# B&R Automation Studio project TD52 (part 110)

#### biogasCyclic.st - Cyclic code
```iecst
(*
***************************************************************************
biogas			control/monitoring gas blower/flare

This code is confidential and proprietary to the INNIO Company.
It may not be used in any form, or reproduced in any manner,
without the express written permission of the INNIO Company.
Copyright, INNIO Company, 2025

Customized modifications: -
------------------------

History:
-------
V0.0		03.12.05/LH	erstellt
V2071		02.02.05/LH	angepasst für V2.071
 			03.03.05/LH	angepasst für neue Gasdrucküberwachungsphilosophie
V2072		16.11.05/LH	angepasst für Modulisierung
V2201		08.08.07/LH	Vorhalte Gasverdichter vor Öffnen 1. Gasstr. während Gasumschaltung
 			12.09.07/LH	Freigabe Fackel nur wenn Gasverdichter nicht gestört ist
V2600		06.08.2009 lettenb.	task activation added
V3.10.0		15.02.2010 lettenb.	QUITT_AB, IN_GT.tAB2GT replaced by reset_alarm[x], quitt_wa
V3.20.0		17.01.2011 lettenb.	connections to alarmsXXxx added, user comment
			14.02.2011	release main gas valve FG_HGV moved to task pb8, enable alarms added
V3.99		21.09.2013	Ganguly/Denk, generated for modular software
V3.99.1		19.09.2013	Denk, V3.30.0 and V3.30.2 changes inserted
V3.99.2		25.03.2013	pankajrodey, Integration for 3.40
V4.03.00	15.03.2016	Denk, Bugfix Alarm Set for A3317
			04.04.2016	Denk, Bugfix Alarm Set for A3328
V4.04.00	26-10-2016	Denk, Logic change for gastemperature messages 3317 and 3568
V4.07.00	19.03.2019	Zengerer, Demand compressor options for TKE Gastrain Types
V4.07.01	16.10.2019	Zengerer, Demand compressor option TOF bMEGA_GasTrain, Operating message: B2997 extended compressor demand for gas leakage check
V4.07.02	25.10.2019	Zengerer  EDGEPOS(OUT_GT.tGT1_SafeDevice.Do) takeover from V4.07 Basisupdate
V4.09.00	16.01.2020	Zengerer  bDelayGDKG_GCStarting to delay leakage check, to allow gas compressor generate sufficient pressure, bDem_SafeDevice	(corr.Jan2020)
			06.02.2020	Zengerer  bMsg2997_Set changed, avaid  GC restart after failure reset
V4.25.00	17.12.2025	Tinello   Safety signals added

Instructions for use:
--------------------
 - activate task if used (see comment)
 - disable gas blower if not existing
 - RM "Fackel in Betrieb" in fb31_hb einbinden und in BILD_50 zur Anzeige bringen!

enable biogas alarms in the specific network if used:			default:

A3316	Gas compressor failure					active
W3567	Gas compressor failure					not active

A3317	Gas temperature high					active
W3568	Gas temperature high					not active
A3328 	Gas temperature measuring signal failure				not active

A3318	Gas pressure low before compressor				active
W3569	Gas pressure low before gas compressor				not active
A3327	Gas pressure before gas compressor measuring signal failure		not active
W3570	Gas pressure before gas compressor measuring signal failure		not active

A3326	Idle operation time gas compressor maximum			active

W3520	Flare failure						active

Outstandings:
------------
*********************************************

*)

PROGRAM _CYCLIC

IF NOT Para.bBiogasActive THEN
	bDelayGDKG_GCStarting := FALSE;				(*inactive bigas compressor should not delay  bDelayGDKG_GCStarting leakage check*)
	RETURN;
ELSE

	(* Alarm Set for A3327: Measurement signal error Gas pressure before compressor *)
	bMsg3327_Set := Para.bMsg3327Active AND NOT IN_GT.tPr_GT_Suct.GoodQual AND NOT OUT_GT.bGT2_Select;

	(* Alarm Set for W3570: Measurement signal error Gas pressure before compressor *)
	bMsg3570_Set := Para.bMsg3570Active AND NOT IN_GT.tPr_GT_Suct.GoodQual AND NOT MM2VIS.bMsg3327 AND NOT bMsg3327_Set;

	(* Alarm Set for A3318 Gas pressure minimum before compressor *)
	xTON_FA_ZM_GDMI11.IN := MM2VIS.bMsgDummy_Min_SuctPr OR NOT IN_GT.tPr_GT_MinBefCompr.Di;
	xTON_FA_ZM_GDMI11.PT := T#2s;
	xTON_FA_ZM_GDMI11();
	HM_GDMI11    := xTON_FA_ZM_GDMI11.Q;
	bMsg3318_Set := HM_GDMI11 AND ((FG_GDRUW AND NOT OUT_GT.bGT2_Select) OR bMsg3318_Set);

	(* Alarm Set for W3569 Gas pressure minimum before compressor maximum *)
	bMsg3569_Set := Para.bMsg3569Active
		            AND HM_GDMI11
		            AND NOT MM2VIS.bMsg3318
		            AND NOT bMsg3318_Set
		            AND Para.bGCActive
		            AND (OUT_GT.bGT_TypSwhActive OR OUT_GT.bGT_TypSwhActiveHalt);

	(* Alarm Set for A3328: Measurement signal from "spec_gas"*)
	bMsg3328_Set := Para.bMsg3328Active AND NOT IN_GT.tT_GT.GoodQual AND NOT OUT_GT.bGT2_Select;

	(* Alarm Set for A3317 Gas temperature maximum *)
	bMsg3317_Set := ((GT_MAX AND IN_GT.tT_GT.GoodQual) OR NOT IN_GT.tT_GT_Ok.Di) AND NOT OUT_GT.bGT2_Select;

	(* Alarm Set for W3568: Gas temperature maximum *)
	bMsg3568_Set := Para.bMsg3568Active AND ((GT_MAX AND IN_GT.tT_GT.GoodQual) OR NOT IN_GT.tT_GT_Ok.Di) AND NOT MM2VIS.bMsg3317 AND NOT bMsg3317_Set;

	(* Alarm Set  for A3316: Trip: Gas compressor failure *)
	bMsg3316_Set := NOT IN_GT.tGT_GC_Fail.Di AND NOT OUT_GT.bGT2_Select;

	(* Alarm Set for W3567: Warning: Gas compressor failure *)
	bMsg3567_Set := Para.bMsg3567Active AND NOT IN_GT.tGT_GC_Fail.Di AND NOT MM2VIS.bMsg3316 AND NOT bMsg3316_Set;

	(* Flare failure *)
	bMsg3520_Set := NOT IN_GT.tGT_FlairFail.Di;

	IF (bMEGA_GasTrain) THEN					(*derived from option bit2 = '4' == MEGA Gas Train, for wide pipe dimensions with 2 separate valves 	(V4.07	Requisition- supplied code parts included for MGV) *)
		(* Demand compressor for Module operation *)
		(*-------------------------------------------------------------------------------------*)
		TOF_MEGA_GC.IN := EDGEPOS(NOT IN_GT.bSafetyPLC_Active AND bDem_SafeDevice)  						// V4.07 Basisupdate 2  old: EDGEPOS(OUT_GT.tGT1_SafeDevice.Do);(* SAFETY PLC *)
						  OR	 (	  IN_GT.bSafetyPLC_Active AND IN_GT.tSafetyLoop_Eng.Di AND NOT IN_GT.bSafeOUT_GT1_SD_Dem_PS); 											(* SAFETY PLC *)

		IF IN_GT.tAB2GT.bGnlTrip1 OR  IN_GT.tAB2GT.bGnlTrip2 OR OUT_GT.bMsg1027 THEN 						// OR IN_GT.tAB2GT.bGnlTrip3 THEN
			TOF_MEGA_GC.PT := 0 ;									// V4.09: avoid  GC restart after failure reset
		ELSE
			TOF_MEGA_GC.PT := IN_GT.tCU2GT.tiGT_TestDuration; 		// T#120s;	 (*time for gas compressor / Gas sfety check [s] *)
		END_IF

		TOF_MEGA_GC();
		(*-------------------------------------------------------------------------------------*)
		bDem_GC_M :=   (IN_GT.bEng_Aux_Dem OR (TOF_MEGA_GC.Q AND NOT IN_GT.tGT1_SafeDevOK.Di AND NOT IN_GT.bSafeOUT_GT1_SafeDevOK))	(*gas compressor demand extension*) 	(* SAFETY PLC *)
				AND NOT IN_GT.bMsg1053
				AND NOT IN_GT.bMsg1054
				AND NOT IN_GT.bMsg1031
				AND NOT OUT_GT.bGT2_Select;

		bMsg2997_Set := Para.bGCActive
				AND OUT_GT.tGT_GC_Dem.Do
				AND bDem_GC_M
				AND NOT IN_GT.tEng_Run.Do
				AND NOT IN_GT.bEng_Aux_Dem
				AND NOT IN_GT.tGT1_SafeDevOK.Di ;
				// := 	Para.bGCActive AND  OUT_GT.tGT_GC_Dem.Do  AND TOF_MEGA_GC.Q	; 		(* Megagas Operating message: B2997 gas compressor demand extension - gas leakage test (new in V4.09)*)

	ELSE
		(* Demand compressor for Module operation *)
		bDem_GC_M := IN_GT.bEng_Aux_Dem 							//OLD: gas compressor demand intermediate  ANF_V_M :=
				AND NOT IN_GT.bMsg1053
				AND NOT IN_GT.bMsg1054
				AND NOT IN_GT.bMsg1031
				AND NOT OUT_GT.bGT2_Select;
	END_IF

		(* Demand Flair *)
	ANF_FA :=	IN_GT.tDemFlair.Di AND NOT IN_GT.bMsg1053 AND NOT IN_GT.bMsg1054 AND NOT IN_GT.bMsg1031
	            AND NOT bDem_GC_M AND IN_GT.tFlairRdy.Di AND NOT MM2VIS.bMsg3520;

	(* Release  Flare (only when Gas compressure has not failed *)
	xTON_FG_FA.IN := IN_GT.tGT_GC_Fail.Di ;
	xTON_FG_FA.PT := T#5s;
	xTON_FG_FA();
	OUT_GT.tGT_RelFlair.Do := xTON_FG_FA.Q AND ANF_FA;

	(* Demand gas compressor *)
	ANF_GVD_1				:=	ANF_FA
	           					OR (bDem_GC_M AND (OUT_GT.tGV1_Open.Do OR V_GVD OR NOT IN_GT.tEng_Run.Do));
	OUT_GT.tGT_GC_Dem.Do 	:= FG_HGV AND ANF_GVD_1 AND NOT MM2VIS.bMsg3318 AND NOT MM2VIS.bMsg3221 AND NOT MM2VIS.bMsg3327 AND NOT MM2VIS.bMsg3326 AND NOT MM2VIS.bMsg3316;

	(* Monitoring idle operation time gas compressor maximum *)
	bMsg3326_Set := OUT_GT.tGT_GC_Dem.Do
					AND ((NOT IN_GT.tEng_Run.Do AND bDem_GC_M) OR (OUT_GT.tGT_RelFlair.Do AND NOT IN_GT.tGT_FlareOpMod.Di));

	(* Release gas pressure monitoring (Gas pressure minimum Gas train 1 (p10_1001)) *)
	xTON_FA_GASV1.IN := OUT_GT.tGV1_Open.Do;
	xTON_FA_GASV1.PT := Para.tiGT1_Delay_Mon;			// 5s parameter introduced in V3.30
	xTON_FA_GASV1();

	xTON_FA_T_GDRUW.IN := IN_GT.bEng_Aux_Dem OR ((bDem_SafeDevice OR NOT IN_GT.bSafeOUT_GT1_SafeDevOK) AND OUT_GT.tGT_GC_Dem.Do);	(*Engine Demand OR Gas Safety Check Demand*)	(* SAFETY PLC *)
	xTON_FA_T_GDRUW.PT := Para.tiGT1_Delay_Mon;			// 5s parameter introduced in V3.30
	xTON_FA_T_GDRUW();

	T_GDRUW := (xTON_FA_GASV1.Q AND IN_GT.tEng_Run.Do) OR (xTON_FA_T_GDRUW.Q AND NOT IN_GT.tEng_Run.Do);

	(*generate flag to delay gas leakage checking*)
	xTOFDelayGDKG_GCStarting.IN	:= EDGEPOS(OUT_GT.tGT_GC_Dem.Do AND NOT IN_GT.tGT1_SafeDevOK.Di);  	(*bit to delay leakage check, to allow time for gas compressor building up sufficient pressure*)

	xTOFDelayGDKG_GCStarting(PT:= T#6s);
	bDelayGDKG_GCStarting 	:=xTOFDelayGDKG_GCStarting.Q ;
END_IF;

END_PROGRAM
```

#### biogas.var - Local variables
```iecst
(********************************************************************
 * COPYRIGHT -- INNIO Company
 ********************************************************************
 * Program: biogas
 * File: biogas.var
 * Author: 105051626
 * Created: April 19, 2012
 ********************************************************************
 * Local variables of program biogas
 ********************************************************************)
VAR
	ANF_FA : BOOL := 0; (* Anforderung Fackel *)
	bDem_GC_M : BOOL; (*Intermediate variable for Demand gas compressor*) (*OldName: ANF_V_M*)
	HM_GDMI11 : BOOL; (*Gas pressure minimum before compresssor*)
	ANF_GVD_1 : BOOL; (*Intermediate variable for interlocks of Demand gas compressor*)
	xTON_FA_ZM_GDMI11 : TON;
	xTON_FA_GASV1 : TON;
	xTON_FG_FA : TON;
	xTON_FA_T_GDRUW : TON;
	TOF_MEGA_GC : TOF; (*Gas compressor timer for Mega Gasvalve option*)
	xTOFDelayGDKG_GCStarting : TOF; (*prevent saftey device reaction to low gas pressure*)
END_VAR
```

### Program Logical/Gastrain/bm3_nm3 (IEC) - bm3_mn3

#### bm3_nm3Cyclic.st - Cyclic code
```iecst
(* BERECHNUNG NORMKUBIKMETER-GASVERBRAUCH

VER	Datum/Name	Änderung
V170	21.03.02/LH	erstellt
V172	31.07.02/LH	Gaszähler-Impuls aus pb7 übernommen
					Berechnung Zustandszahl eliminiert => neuer task
		17.09.02/LH	korrigiert für AS 2.2
V173	11.11.02/LH	Vergleich korrigiert
V181	23.04.03/LH	Zähler-Beschaltung richtiggestellt
V190	18.06.04/LH	Vermeidung von Rundungsfehlern
V03.99.00	21.09.2013	Ganguly/Denk 	Generated for modular software
V04.00.02	02.06.2014  Denk			Gas counter to MM2VIS added
V04.01.00	01.07.2014  Denk			Gas counter parameters added and additional OUT-Interfaces
V04.01.01	18.03.2015	lettenb.		increase counter with NORM_IMP, xR_TRIG_FA_BTRB_IMP.Q only for 1 cycle
V04.03.00	02.06.2015	Denk			Bugfix, gas counter reset when PLC coldstart. Connected to Perm struct.
V04.04.00	18.10.2016	Denk			Gas counter writable from Visu
V04.07.00	10.04.2019	Zengerer		Gas counter prescaler for requisition demanded version V4.07, chapter 5
V04.07.01	11.04.2019	Zengerer		xTOF_FA_BTRB_M3.PT := ...tiGCPulse_Duration_min
V04.07.02	05.06.2019	Zengerer		cleanup, disabeled xCTD_FA_GAS_IMP removed

Instructions FOR use:
--------------------
 -

Outstandings:
------------
rGasImp_Prescaling < 1.0 ..  //TODO:Release after pilot engines in V4.09

**********************************************)

PROGRAM _CYCLIC

    (* Reset Nm3-Impulse *)
	NORM_IMP := FALSE;

	(* Gas counter - impulse *)

	IF IN_GT.tCU2GT.iGC_Select_Option.7  THEN 					// Bit 7 sets task input back to behavior of former task version <4.07
		xR_TRIG_FA_GAS_IMP_CD.CLK := IN_GT.tCnt_GasImp.Di;		// Direct DI input like in former task version <4.07
	ELSE
		xR_TRIG_FA_GAS_IMP_CD.CLK := bGasImp_Prescaled;			// Pulse prescaler for IN_GT.tCnt_GasImp.Di gets handled in TC2
	END_IF
	xR_TRIG_FA_GAS_IMP_CD();
	IF NOT IN_GT.tCnt_GasImp.Di THEN bGasImp_Prescaled := FALSE; END_IF	(* Do not clear the artificial generated pulse, until the real pulse is gone, to keep similar pulse duration behavior *)

	BTRB_IMP   := xR_TRIG_FA_GAS_IMP_CD.Q AND ANLAUF;

	ANLAUF := TRUE;											// Setting local flag to TRUE , it is initially FALSE

	(* Bm3-Impulse *)
	xTOF_FA_BTRB_M3.IN := BTRB_IMP;
	xTOF_FA_BTRB_M3.PT := IN_GT.tCU2GT.tiGCPulse_Duration_min ;   		// := T#1s;
	xTOF_FA_BTRB_M3();
	BTRB_M3 := xTOF_FA_BTRB_M3.Q;

	(* Edge triggered Gas count impulse *)
	xR_TRIG_FA_BTRB_IMP.CLK := BTRB_M3;
	xR_TRIG_FA_BTRB_IMP();

	IMP_W := LIMIT(1000, Para.rGasImp_Prescaling * 1000, 50000);		 (*NEW parameter from V4.07: (Impulswertigkeit (Caution: formerly Constant value 1000 removed, but 1000 has to be FIXED LOWER LIMIT to cooperate with prescaler!)  *)

	IF xR_TRIG_FA_BTRB_IMP.Q THEN
		IMP_B := IMP_W;
	ELSE
		IMP_B := 0;
	END_IF;

	(* L10-L12 Summe *)
	IMP_N := ZSZ * IMP_B;

	(* Sum up impulses *)
	IMP_S := LIMIT(0, (IMP_S + IMP_N) ,4294967295);

	(* Block new impulse *)
	xTOF_FA_T_NORM_M3.IN := NORM_M3;
	xTOF_FA_T_NORM_M3.PT := IN_GT.tCU2GT.tiGCPulse_Duration_min ;   		// := T#1s;
	xTOF_FA_T_NORM_M3();
	T_NORM_M3 := xTOF_FA_T_NORM_M3.Q;

	(* Sum greater than impulse "wertigkeit" & release new impulse *)
	IF ((IMP_S >= IMP_W) AND NOT T_NORM_M3) THEN
		(* Set Nm3 impulse *)
		NORM_IMP := TRUE;
		(* Reduce sum by impulse "wertigkeit *)
		IMP_S := IMP_S - IMP_W;
	END_IF;

	(* Nm3 impulse *)
	xTOF_FA_NORM_M3.IN := NORM_IMP;
	xTOF_FA_NORM_M3.PT := IN_GT.tCU2GT.tiGCPulse_Duration_min ;   		// := T#1s;
	xTOF_FA_NORM_M3();
	NORM_M3 := xTOF_FA_NORM_M3.Q;

	(* Counter *)
	IF Para.bCnt_Gas_NormM3 THEN
		(* Gas counter Norm_M3 *)
		IF NORM_IMP THEN
			(* increase counter *)
			MM2VIS.iCnt_Gas_NormM3 := MM2VIS.iCnt_Gas_NormM3 + REAL_TO_DINT(MAX(1, Para.rGasImp_Prescaling));  // + 1; 	 Changed V4.07
			(* check limits *)
		ELSIF MM2VIS.iCnt_Gas_NormM3 >= 1000000000 THEN
			MM2VIS.iCnt_Gas_NormM3 := MM2VIS.iCnt_Gas_NormM3 - 1000000000;    (* check upper limit *)
		ELSIF MM2VIS.iCnt_Gas_NormM3 <= -1000000000 THEN
			MM2VIS.iCnt_Gas_NormM3 := MM2VIS.iCnt_Gas_NormM3 + 1000000000;    (* check lower limit *)
		END_IF;
	END_IF;

	IF Para.bCnt_Gas_OpM3 THEN
		(* Gas counter Op_M3 *)
		IF xR_TRIG_FA_BTRB_IMP.Q THEN
			(* increase counter *)
			MM2VIS.iCnt_Gas_OpM3 := MM2VIS.iCnt_Gas_OpM3 + REAL_TO_DINT(MAX(1, Para.rGasImp_Prescaling));  // + 1; 	 Changed V4.07
			(* check limits *)
		ELSIF MM2VIS.iCnt_Gas_OpM3 >= 1000000000 THEN
			MM2VIS.iCnt_Gas_OpM3 := MM2VIS.iCnt_Gas_OpM3 - 1000000000;        (* check upper limit *)
		ELSIF MM2VIS.iCnt_Gas_OpM3 <= -1000000000 THEN
			MM2VIS.iCnt_Gas_OpM3 := MM2VIS.iCnt_Gas_OpM3  + 1000000000;       (* check lower limit *)
		END_IF;
	END_IF;

	(* Assignement to OUT/MM2VIS-Interfaces *)
	OUT_GT.iCnt_Gas_OpM3   	:= MM2VIS.iCnt_Gas_OpM3;
	OUT_GT.iCnt_Gas_NormM3 	:= MM2VIS.iCnt_Gas_NormM3;
	OUT_GT.bCnt_Gas_OpM3   	:= BTRB_M3;
	OUT_GT.bCnt_Gas_NormM3 	:= NORM_M3;

END_PROGRAM
```

#### bm3_nm3.var - Local variables
```iecst
VAR
	ANLAUF : BOOL := 0;
	BTRB_IMP : BOOL := 0;
	BTRB_M3 : BOOL; (*Bm3 impulse   	CV_GAS_IMP : UINT := 0;	*)
	IMP_B : REAL;
	IMP_N : REAL;
	IMP_S : REAL; (* Impulssumme *)
	IMP_W : REAL; (* 1000 Impulswertigkeit (Caution: parameter value from V4.07 onward)*)
	NORM_IMP : BOOL;
	NORM_M3 : BOOL;
	T_NORM_M3 : BOOL := 0;  (*	xCTD_FA_GAS_IMP : CTD;  *)
	xR_TRIG_FA_BTRB_IMP : R_TRIG;
	xR_TRIG_FA_GAS_IMP_CD : R_TRIG;  (*	xR_TRIG_FA_GAS_IMP_LD : R_TRIG; *)
	xTOF_FA_BTRB_M3 : TOF;
	xTOF_FA_NORM_M3 : TOF;
	xTOF_FA_T_NORM_M3 : TOF;
END_VAR
```

### Program Logical/Gastrain/spec_gas (IEC) - spec_gas

#### spec_gasCyclic.st - Cyclic code
```iecst
(* MONITORING AND CONTROLING OF SPECIAL GAS ENGINES

variables (limit switches) for customized use:
 	GD_MAX	gas pressure maximum
 	GT_MAX	gas temperature maximum
 	GT_MIN	gas temperature minimum
 	SD_MAX	suction pressure maximum
 	SD_MIN	suction pressure minimum

MS_CV calorific value measuring signal failure
CV_MIN_A calorific value low
CV_MIN_W calorific value low
CV_RED reduction by calorific value active
OUT_GT.rP_Red_CV_Norm reduction value by calorific value

output variables to standard software:

BOOL:	CH4_MIN_A	--> A1086
 	CH4_MIN_W	--> W3154
 	FGGAS		--> W3153
 	GD_MIN_W	--> W3221
 	MS_CH4		--> W3155
 	MS_GD		--> W3156
 	MS_GM		--> W3160
 	MS_GT		--> W3159
 	MS_O2_A 	--> A1088
 	MS_O2_W 	--> W3158
 	MS_SD		--> W3157
 	O2_MAX		--> A1087

............................
VER	Datum/Name	Änderung
V180	19.11.02/LH	erstellt
V181	10.04.03/Th.	Korrekturen bei Typprüfung: OUT_GT.bGasSupplyOk
 	    11.04.03/Th.	Korrekturen bei Typprüfung: MS_O2_W, MS_O2_A
 	    17.04.03/Th.	Korrekturen bei Typprüfung: SD_MIN, SD_MAX
V183	16.10.03/LH	Messignal CH4-Gehalt erst aktiv mit IN_GT.bParaSetupOk
V184	07.01.04/ThJ	Messignalstörungen erst aktiv mit IN_GT.bParaSetupOk;
 			Reset CH4_MIN, MS_GM, MS_O2_A, MS_O2_W wenn nicht aktiviert.
 			Kommentare.
 			Zeitverz. für CH4_MIN 2 --> 5s.
V2071	30.11.04/LH	Korrektur Gasqualitätsberechnung
 	    03.02.05/LH	Überwachung Gasdruck minimum angepasst für V2071
 	    03.03.05/LH	Anpassung Saugdruck min/max
V2072	16.11.05/LH	CH4 min. / Gasdr. min. / Freigabe aus Gasstation lt. letzten Erkenntnissen angepasst
 			     Anforderung Entlastung eliminiert (wird nicht benötigt)
V190	19.03.04/LH	Interpolation GAS1_2 über Rezept einstellbar
 		    	 Leistungsreduktionen --> p_soll(classic)/powersel(XT)
 			     Umrechnungen --> ana_umr(classic)/ana_calc(XT)
V220	19.02.07/LH	angepasst für X20-Einführung
 	    01.03.07/LH	Erweiterung auf Pt100
 	    10.04.07/LH	Zuweisung für Pt100
V2.32	14.07.08/ThJ Heizwert/calorific value added
V2.34.0 04.12.2008 Lett./ThJ set GAS1_2 in case of Para.bGT_CVIpol12Active=true
V2.50.0	02.02.2009 lett. HW_WE -> AI_CV(for standard)
V03.99.00.00	21.09.2013	Ganguly	generated for modular software
V03.99.01.00	21.02.2013	Denk	Integration of V3.30 in modular software
									HM_GDMI1, HM_GDMI2 changed to modul global variable
V04.00.02.00	15.05.2014	Denk	Bugfix, FGGAS
V04.00.02.00	17.05.2014	Denk	Bugfix, Interpolations-Umschaltung, 4x Skalierung falsch 100% --> 1.0%
V04.01.00.00	17.07.2014	Denk	Bugfix, Measurement signal failure reset CH4 and CV signal
									Bugfix, Deactivation power reduction (CH4,GD,SD) via standard DI's
									Bugfix, CH4,CV: Para.rGT_CH4Mix1,Para.rGT_CH4Mix2 and Para.bGT_CVIpol12Active
V04.01.01.00	24.08.2014	Denk	Bugfix, Interpolation deactivation
V04.01.02.00	14.10.2014	Denk	Bugfix, Message activation O2 max.
V04.03.00.00	31.03.2015	Denk	Improvement, additional LABELS for tPr_GT1_1_Min and tPr_GT1_1_Max
				02.07.2015	Denk 	Bugfix, 3221 not activ when gastrain 2 is active. NOT was missing. NOT MM2VIS.bMsg1028
									Warnings for 4 gaslines bMsg2694-2696 added
V04.10.0.00		08.12.2020	Denk	Bugfix, xTON_GDMA2() changed to xTON_GDMA2_VISA()
         		10.12.2020	Zuschnig	Included power reduction for Tecjet differential pressure
				21.01.2020	Zuschnig	Bugfix, Power reduction suction pressure (swap X1<->X2)
V04.11.0.00		02.03.2022	Zuschnig	Include CH4 signal via Bus from customize modul
V04.12.0.00		22.01.2023	Zuschnig	Include H2 signal processing, power reduction and limit detection
V04.13.0.00		26.05.2023	Zuschnig	Include measuring signal failure setpoint - Gas mixing
*)
PROGRAM _INIT
	(*Parameter*)
	SimPID_deltaP_TJ.P 			:= 0.001;
	SimPID_deltaP_TJ.I 			:= 0;
	SimPID_deltaP_TJ.D			:= 0;
	SimPID_deltaP_TJ.N			:= 0;
	SimPID_deltaP_TJ.wxmax		:= 0.2; (* maximum 200mbar delta P *)
	SimPID_deltaP_TJ.wxmin		:= 0;
	SimPID_deltaP_TJ.umax 		:= 0;
	SimPID_deltaP_TJ.umin 		:= -0.5; (* maximum power reduction 50% *)
	SimPID_deltaP_TJ.Kt			:= 1;
	SimPID_deltaP_TJ.deadband 	:= 0.001; (* 1mbar deadband *)
	SimPID_deltaP_TJ.invert 	:= TRUE;

	(*Input*)
	SimPID_deltaP_TJ.u_man		:=	0;
	SimPID_deltaP_TJ.a			:= 	0;
	SimPID_deltaP_TJ.reset		:=  FALSE;
	SimPID_deltaP_TJ.I0			:=  0;
	SimPID_deltaP_TJ.D0			:=  0;
	SimPID_deltaP_TJ.fbk_mode	:=  2;
	SimPID_deltaP_TJ.u_fbk		:=  0;
END_PROGRAM

PROGRAM _CYCLIC
	(* H2 measurement *)
	(* Hand over filtered H2 value *)
	OUT_GT.rH2		:= xLCRPT1_H2.y;
	(* H2 value for H2 compensation of ITP and boost pressure *)
	xGR_MAXR_H2_Comp(In:= OUT_GT.rH2, Gw:= rGwH2_Comp, Hy:= rHyH2_Comp);
	IF xGR_MAXR_H2_Comp.Q THEN
		OUT_GT.rH2_Comp := MAX(0.02, MIN(0.25, OUT_GT.rH2));
	ELSE
		OUT_GT.rH2_Comp := 0;
	END_IF;

	IF Para.bGT_H2Active THEN
		(* Power reduction H2 content *)
		(* Power reduction measurement signal failure H2 content *)
		IF bS_MSF_H2 THEN
			rReductionPowerH2_MSF := Para.rP_Red_H2_MSF;
		ELSE
			rReductionPowerH2_MSF := 1.00;
		END_IF;

		(* Power reduction H2 content high *)
		IF OUT_GT.rH2 > Para.rP_Red_H2Start THEN
			rReductionPowerH2 := 1.00 - ((OUT_GT.rH2 - Para.rP_Red_H2Start) * Para.rP_Red_H2_Rate * 100);
		ELSE
			rReductionPowerH2 := 1.00;
		END_IF;

		OUT_GT.rP_Red_H2_Norm := MIN(rReductionPowerH2_MSF, rReductionPowerH2);

		(* H2 content maximum warning *)
		xGR_MAXR_FA_H2_MAX_W.In := OUT_GT.rH2;
		xGR_MAXR_FA_H2_MAX_W.Gw	:= Para.rGT_H2WarnLimMax;
		xGR_MAXR_FA_H2_MAX_W.Hy := 0;
		xGR_MAXR_FA_H2_MAX_W();

		bH2_MAX_W	:= xGR_MAXR_FA_H2_MAX_W.Q AND IN_GT.tPB2MM.bParaSetupOk;

		(* H2 content maximum alarm *)
		xGR_MAXR_FA_H2_MAX_A.In := OUT_GT.rH2;
		xGR_MAXR_FA_H2_MAX_A.Gw	:= Para.rGT_H2TripLimMax;
		xGR_MAXR_FA_H2_MAX_A.Hy := 0;
		xGR_MAXR_FA_H2_MAX_A();

		bH2_MAX_A	:=	xGR_MAXR_FA_H2_MAX_A.Q AND IN_GT.tPB2MM.bParaSetupOk;
	ELSE
		OUT_GT.rP_Red_H2_Norm	:= 1.00;
		rReductionPowerH2_MSF 	:= 1.00;
		rReductionPowerH2 		:= 1.00;
		bH2_MAX_W				:= FALSE;
		bH2_MAX_A				:= FALSE;
	END_IF;

	(*************************************************************************************************************)
	(* CH4 measurement *)

	IF Para.bGT_CH4Active THEN
		(* Measurement signal failure CH4 content  W3155 !!!!! Alarm not is list *)
		MS_CH4 := NOT IN_GT.tGT_CH4.GoodQual AND IN_GT.tPB2MM.bParaSetupOk AND NOT IN_GT.bCH4_Bus_Active;

		(* Messignalstörung *)
		(* Measurement signal failure *)
		S_MS_CH4 := MS_CH4 OR (S_MS_CH4 AND NOT IN_GT.tAB2GT.bResetWarning );

		(* Hold analog value during calibration *)
		IF IN_GT.tGT_CalibrateActive.Di OR IN_GT.bGT_CalibrateActive_Bus THEN
			rGT_CH4 := rGT_CH4;
		ELSIF NOT IN_GT.bCH4_Bus_Active THEN
			rGT_CH4 := IN_GT.tGT_CH4.Ai;
		ELSE
			rGT_CH4 := IN_GT.rCH4_Bus;
		END_IF;

		(* Reduction due to CH4 content *)
		RED_CH4_a := Para.bP_Red_CH4Active AND NOT MS_CH4 AND NOT IN_GT.tP_Red_CH4Active.Di AND IN_GT.tPB2MM.bParaSetupOk;

		IF RED_CH4_a THEN
			xSigScalR_FA_CH4_RED.X  := rGT_CH4;
			xSigScalR_FA_CH4_RED.X1 := Para.rP_Red_CH4HalfLoad;
			xSigScalR_FA_CH4_RED.Y1 := 0.50;
			xSigScalR_FA_CH4_RED.X2 := Para.rP_Red_CH4Start;
			xSigScalR_FA_CH4_RED.Y2 := 1.00;
			xSigScalR_FA_CH4_RED();
			OUT_GT.rP_Red_CH4_Norm := LIMIT(0.50,xSigScalR_FA_CH4_RED.Y_SCAL,1.000);
		ELSE
			OUT_GT.rP_Red_CH4_Norm := 1.0;
		END_IF;

		(* CH4-Gehalt minimum Warnung/Blockierung (W3154) *)
		CH4_MIN_W_a := Para.bGT_CH4WarnActive AND NOT MS_CH4;

		xGR_MINR_FA_CH4_MIN_W.In := rGT_CH4;
		xGR_MINR_FA_CH4_MIN_W.Gw := Para.rGT_CH4WarnLimMin;
		xGR_MINR_FA_CH4_MIN_W.Hy := Para.rGT_CH4WarnHyMin;
		xGR_MINR_FA_CH4_MIN_W();
		xTON_FA_T_CH4_W.IN := xGR_MINR_FA_CH4_MIN_W.Q AND IN_GT.tPB2MM.bParaSetupOk;
		xTON_FA_T_CH4_W.PT := T#5s;
		xTON_FA_T_CH4_W();
		CH4_MIN := xTON_FA_T_CH4_W.Q AND CH4_MIN_W_a;

		xTON_FA_CH4_MIN.IN := (IN_GT.bEng_Aux_Dem OR CH4_MIN_W) AND NOT OUT_GT.bGT2_Select AND CH4_MIN AND (IN_GT.iIdx_OMSS = 2);
		IF bTestEnabled THEN
			xTON_FA_CH4_MIN.PT := T#3s;
		ELSE
			xTON_FA_CH4_MIN.PT := T#300s;
		END_IF;
		xTON_FA_CH4_MIN();

		CH4_MIN_W_1 := CH4_MIN AND (IN_GT.iIdx_OMSS = 2) AND xTON_FA_CH4_MIN.Q;
		CH4_MIN_W   := (IN_GT.bEng_Aux_Dem OR CH4_MIN_W) AND NOT OUT_GT.bGT2_Select AND (CH4_MIN OR CH4_MIN_W_1);

		(* CH4-Gehalt minimum Abstellung (A1086) *)
		(* CH4-content minimum Trip A1086 *)
		xGR_MINR_FA_CH4_MIN_A.In := rGT_CH4;
		xGR_MINR_FA_CH4_MIN_A.Gw := Para.rGT_CH4TripLimMin;
		xGR_MINR_FA_CH4_MIN_A.Hy := Para.rGT_CH4TripHyMin;
		xGR_MINR_FA_CH4_MIN_A();
		xTON_FA_T_CH4_A.IN := xGR_MINR_FA_CH4_MIN_A.Q AND IN_GT.tPB2MM.bParaSetupOk;
		xTON_FA_T_CH4_A.PT := T#0.5s;
		xTON_FA_T_CH4_A();
		CH4_MIN_A := xTON_FA_T_CH4_A.Q AND Para.bGT_CH4TripActive;
	ELSE
		MS_CH4 	  := FALSE;
		S_MS_CH4  := FALSE;
		CH4_MIN   := FALSE;
		CH4_MIN_W := FALSE;
		CH4_MIN_A := FALSE;
		OUT_GT.rP_Red_CH4_Norm := 1.0;
	END_IF;

	(*************************************************************************************************************)
	(* Heating value *)
	// L20,21 shifted out to HAL IO
	IF Para.bGT_CVActive THEN
		(* Measuring signal failure of heating value *)
		MS_CV   := IN_GT.tPB2MM.bParaSetupOk AND NOT IN_GT.tGT_CV.GoodQual AND NOT IN_GT.bCV_Bus_Active;
		S_MS_CV := MS_CV OR (S_MS_CV AND NOT IN_GT.tAB2GT.bResetWarning );

		(* Hold analog value during calibration *)
		IF IN_GT.tGT_CalibrateActive.Di OR IN_GT.bGT_CalibrateActive_Bus THEN
			rGT_CV := rGT_CV;
		ELSIF NOT IN_GT.bCV_Bus_Active THEN
			rGT_CV := IN_GT.tGT_CV.Ai;
		ELSE
			rGT_CV := IN_GT.rCV_Bus;
		END_IF;

		(* Power reduction due to heat value L25 *)
		RED_CV_a := Para.bP_Red_CVActive AND NOT MS_CV AND NOT CVRED_0 AND IN_GT.tPB2MM.bParaSetupOk;

		xSigScal_FA_CV_RED.X  := rGT_CV;
		xSigScal_FA_CV_RED.X1 := Para.rP_Red_CVHalfLoad;
		xSigScal_FA_CV_RED.Y1 := 0.50;
		xSigScal_FA_CV_RED.X2 := Para.rP_Red_CVStart;
		xSigScal_FA_CV_RED.Y2 := 1.00;
		xSigScal_FA_CV_RED();

		IF RED_CV_a THEN
			OUT_GT.rP_Red_CV_Norm := LIMIT(0.00,xSigScal_FA_CV_RED.Y_SCAL,1.00);
		ELSE
			OUT_GT.rP_Red_CV_Norm := 1.0;
		END_IF;

		(* Heizwert minimum Warnung/Blockierung (Wxxxx) *)
		(* Calorific value Warning/Blocking (Wxxxx) *)
		CV_MIN_W_a := Para.bGT_CVWarnActive AND NOT MS_CV;

		xGR_MINR_FA_CV_MIN_W.In := IN_GT.tGT_CV.Ai;
		xGR_MINR_FA_CV_MIN_W.Gw := Para.rGT_CVWarnLimMin;
		xGR_MINR_FA_CV_MIN_W.Hy := Para.rGT_CVWarnHyMin;
		xGR_MINR_FA_CV_MIN_W();
		xTON_FA_T_CV_W.IN := xGR_MINR_FA_CV_MIN_W.Q AND IN_GT.tPB2MM.bParaSetupOk;
		xTON_FA_T_CV_W.PT := T#5s;
		xTON_FA_T_CV_W();
		CV_MIN := xTON_FA_T_CV_W.Q AND CV_MIN_W_a;

		xTON_FA_CV_MIN.IN := (IN_GT.bEng_Aux_Dem OR bMsg_Dummy_Warn_CV) AND NOT OUT_GT.bGT2_Select AND CV_MIN AND (IN_GT.iIdx_OMSS = 2);
		IF bTestEnabled THEN
			xTON_FA_CV_MIN.PT := T#3s;
		ELSE
			xTON_FA_CV_MIN.PT := T#300s;
		END_IF;
		xTON_FA_CV_MIN();

		// CV_MIN_W -> Warning: calorific value minimum
		bMsg_Dummy_Warn_CV := xTON_FA_CV_MIN.Q OR (CV_MIN AND NOT OUT_GT.bGT2_Select AND (IN_GT.bEng_Aux_Dem OR bMsg_Dummy_Warn_CV));

		(* Heizwert minimum Abstellung (Axxxx) *)
		(* Calorific value minimum Trip (Axxx) *)
		xGR_MINR_FA_CV_MIN_A.In := IN_GT.tGT_CV.Ai;
		xGR_MINR_FA_CV_MIN_A.Gw := Para.rGT_CVTripLimMin;
		xGR_MINR_FA_CV_MIN_A.Hy := Para.rGT_CVTripHyMin;
		xGR_MINR_FA_CV_MIN_A();
		xTON_FA_T_CV_A.IN := xGR_MINR_FA_CV_MIN_A.Q AND IN_GT.tPB2MM.bParaSetupOk;
		xTON_FA_T_CV_A.PT := T#0.5s;
		xTON_FA_T_CV_A();
		// CV_MIN_A -> Trip: calorific value minimum
		bMsg_Dummy_Trip_CV := xTON_FA_T_CV_A.Q AND Para.bGT_CVTripActive;

	ELSIF NOT Para.bGT_CVActive THEN
		MS_CV                 := FALSE;
		S_MS_CV               := FALSE;
		CV_MIN                := FALSE;
		bMsg_Dummy_Warn_CV    := FALSE;
		bMsg_Dummy_Trip_CV    := FALSE;
		OUT_GT.rP_Red_CV_Norm := 1.0;
		rP_Red_CV_Norm        := 1.0;
	END_IF;

	(*****************************************************************************************************************)
	(* 	activate interpolation gas1 & gas2 (set: GAS1_2 = parameter interpolation gas1 & 2 active):
	if:
	Para.bGT_CVActive        = true: parameter calorific value active, (interpolation from CV is priority)
	and Para.bGT_SpecGasActive = true: parameter special gas active
	and Para.bGT_CVIpol12Active   = true: parameter interpolation active from CV  *)

	OUT_GT.bGT_Ipol12Active := FALSE;

	IF 	(NOT Para.bGT_CVActive OR NOT Para.bGT_SpecGasActive) THEN			//old code: weiter0 Bedingung erfüllt
		IF ((NOT Para.bGT_Ipol12Active_Para OR NOT Para.bGT_CH4Active ) AND
			(NOT Para.bGT_CVIpol12Active OR NOT Para.bGT_CVActive) OR
			NOT Para.bGT_SpecGasActive) THEN
			// weiter0:
			X_GMISCH_2 := 0.0;												//old code: weiter1 Bedingung erfüllt
		ELSE
			IF (Para.bGT_CVIpol12Active AND Para.bGT_CVActive) THEN
				// L043
				// X_GMISCH_2_CalVal
				xSigScal_R_FA_CalVal_GMV.X  := LIMIT(Para.rGT_CV4Mix1, rGT_CV, Para.rGT_CV4Mix2);
				xSigScal_R_FA_CalVal_GMV.X1 := Para.rGT_CV4Mix1;
				xSigScal_R_FA_CalVal_GMV.Y1 := 0.0;
				xSigScal_R_FA_CalVal_GMV.X2 := Para.rGT_CV4Mix2;
				xSigScal_R_FA_CalVal_GMV.Y2 := 1.0;
				xSigScal_R_FA_CalVal_GMV();
				Y_SCAL_CalVal := xSigScal_R_FA_CalVal_GMV.Y_SCAL;

				IF (NOT Para.bGT_CVActive OR S_MS_CV) THEN
					X_GMISCH_2 := Para.rGT_CV_Mix_DefVal;
				ELSE
					X_GMISCH_2 := Y_SCAL_CalVal;
				END_IF;

				OUT_GT.bGT_Ipol12Active := Para.bGT_CVIpol12Active;

			ELSE
				// L040
				// Mixed gas relation from CH4-content
				xSigScalR_FA_CH4_GMV.X  := LIMIT(Para.rGT_CH4Mix1,rGT_CH4,Para.rGT_CH4Mix2);
				xSigScalR_FA_CH4_GMV.X1 := Para.rGT_CH4Mix1;
				xSigScalR_FA_CH4_GMV.Y1 := 0.0;
				xSigScalR_FA_CH4_GMV.X2 := Para.rGT_CH4Mix2;
				xSigScalR_FA_CH4_GMV.Y2 := 1.0;
				xSigScalR_FA_CH4_GMV();

				IF (NOT Para.bGT_CH4Active OR S_MS_CH4) THEN
					X_GMISCH_2 := Para.rGT_CH4_Mix_DefVal;
				ELSE
					X_GMISCH_2 := xSigScalR_FA_CH4_GMV.Y_SCAL;
				END_IF;

				OUT_GT.bGT_Ipol12Active := Para.bGT_Ipol12Active_Para;

			END_IF;
		END_IF;
	ELSE
		IF ((NOT Para.bGT_Ipol12Active_Para OR NOT Para.bGT_CH4Active) AND
			(NOT Para.bGT_CVIpol12Active OR NOT Para.bGT_CVActive) OR
			NOT Para.bGT_SpecGasActive) THEN
			// weiter0:
			X_GMISCH_2 := 0.0;												//old code: weiter1 Bedingung erfüllt
		ELSE
			IF (Para.bGT_CVIpol12Active AND Para.bGT_CVActive) THEN
				// L043
				// X_GMISCH_2_CalVal
				xSigScal_R_FA_CalVal_GMV.X  := LIMIT(Para.rGT_CV4Mix1, rGT_CV, Para.rGT_CV4Mix2);
				xSigScal_R_FA_CalVal_GMV.X1 := Para.rGT_CV4Mix1;
				xSigScal_R_FA_CalVal_GMV.Y1 := 0.0;
				xSigScal_R_FA_CalVal_GMV.X2 := Para.rGT_CV4Mix2;
				xSigScal_R_FA_CalVal_GMV.Y2 := 1.0;
				xSigScal_R_FA_CalVal_GMV();
				Y_SCAL_CalVal := xSigScal_R_FA_CalVal_GMV.Y_SCAL;

				IF (NOT Para.bGT_CVActive OR S_MS_CV) THEN
					X_GMISCH_2 := Para.rGT_CV_Mix_DefVal;
				ELSE
					X_GMISCH_2 := Y_SCAL_CalVal;
				END_IF;

				OUT_GT.bGT_Ipol12Active := Para.bGT_CVIpol12Active;

			ELSE
				// L040
				// Mixed gas relation from CH4-content
				xSigScalR_FA_CH4_GMV.X  := LIMIT(Para.rGT_CH4Mix1,rGT_CH4,Para.rGT_CH4Mix2);
				xSigScalR_FA_CH4_GMV.X1 := Para.rGT_CH4Mix1;
				xSigScalR_FA_CH4_GMV.Y1 := 0.0;
				xSigScalR_FA_CH4_GMV.X2 := Para.rGT_CH4Mix2;
				xSigScalR_FA_CH4_GMV.Y2 := 1.0;
				xSigScalR_FA_CH4_GMV();

				IF (NOT Para.bGT_CH4Active OR S_MS_CH4) THEN
					X_GMISCH_2 := Para.rGT_CH4_Mix_DefVal;
				ELSE
					X_GMISCH_2 := xSigScalR_FA_CH4_GMV.Y_SCAL;
				END_IF;

				OUT_GT.bGT_Ipol12Active := Para.bGT_Ipol12Active_Para;

			END_IF;
		END_IF;
	END_IF;

	MM2VIS.bGT_Ipol12Active := OUT_GT.bGT_Ipol12Active;

	(* Gas pressure *)
	IF Para.bPr_GT_GasPrActive THEN
		MS_GD := IN_GT.tPB2MM.bParaSetupOk AND NOT IN_GT.tPr_GT_Gas.GoodQual;
		RED_GD_a := Para.bP_Red_GasPrActive AND NOT MS_GD AND NOT IN_GT.tP_Red_GasPrActive.Di AND IN_GT.tPB2MM.bParaSetupOk;

		IF RED_GD_a THEN
			xSigScalR_FA_GD_RED.X  := IN_GT.tPr_GT_Gas.Ai;
			xSigScalR_FA_GD_RED.X1 := Para.rP_Red_GasPrStart;
			xSigScalR_FA_GD_RED.Y1 := 1.00;
			xSigScalR_FA_GD_RED.X2 := Para.rP_Red_GasPrHalfLoad;
			xSigScalR_FA_GD_RED.Y2 := 0.50;
			xSigScalR_FA_GD_RED();
			OUT_GT.rP_Red_GasPr_Norm := xSigScalR_FA_GD_RED.Y_SCAL;
		ELSE
			OUT_GT.rP_Red_GasPr_Norm := 1.0;
		END_IF;

		(* W3221 Gas pressure minimum warning/blocking gas train 1 *)
		GD_MIN_a := Para.bPr_GT_MinActive AND IN_GT.tPr_GT_Gas.GoodQual;

		xGR_MIN_FA_GD_MIN.In := IN_GT.tPr_GT_Gas.Ai;
		xGR_MIN_FA_GD_MIN.Gw := Para.rPr_GT_LimMin;
		xGR_MIN_FA_GD_MIN.Hy := Para.rPr_GT_HyMin;
		xGR_MIN_FA_GD_MIN();
		GD_MIN := xGR_MIN_FA_GD_MIN.Q AND GD_MIN_a;

		ZM := (FG_GDRUW OR (GD_MIN_W AND NOT Para.bGCActive)) AND
		NOT OUT_GT.bGT2_Select AND
		(T_GDRUW OR NOT Para.bGCActive);

		xTP_FA_GD_MIN_W.IN := ZM AND GD_MIN AND (IN_GT.iIdx_OMSS = 2);
		// Timer duration modified for testing
		IF bTestEnabled THEN
			xTP_FA_GD_MIN_W.PT := T#3s;
		ELSE
			xTP_FA_GD_MIN_W.PT := T#300s;
		END_IF;
		xTP_FA_GD_MIN_W();
		GD_MIN_W := xTP_FA_GD_MIN_W.Q OR (ZM AND GD_MIN);

		bMsg3221_Set := GD_MIN_W OR
		(HM_GDMI1 AND NOT MM2VIS.bMsg1028 AND NOT Para.bGCActive AND
		(OUT_GT.bGT_TypSwhActive OR OUT_GT.bGT_TypSwhActiveHalt));

		(* W2694 Gas pressure minimum warning/blocking gas train 1 line 2 *)
		bMsg2694_Set := HM_GDMI1_2 AND NOT MM2VIS.bMsg1028 AND NOT Para.bGCActive AND
		(OUT_GT.bGT_TypSwhActive OR OUT_GT.bGT_TypSwhActiveHalt);

		(* W2695 Gas pressure minimum warning/blocking gas train 1 line 3 *)
		bMsg2695_Set := HM_GDMI1_3 AND NOT MM2VIS.bMsg1028 AND NOT Para.bGCActive AND
		(OUT_GT.bGT_TypSwhActive OR OUT_GT.bGT_TypSwhActiveHalt);

		(* W2696 Gas pressure minimum warning/blocking gas train 1 line 4 *)
		bMsg2696_Set := HM_GDMI1_4 AND NOT MM2VIS.bMsg1028 AND NOT Para.bGCActive AND
		(OUT_GT.bGT_TypSwhActive OR OUT_GT.bGT_TypSwhActiveHalt);

		(* W3222 Gas pressure minimum gas train 2 *)
		bMsg3222_Set := HM_GDMI2 AND NOT MM2VIS.bMsg1030;

		(* Gas pressure maximum *)
		GD_MAX_a := Para.bPr_GT_MaxActive AND IN_GT.tPr_GT_Gas.GoodQual;

		xGR_MAX_FA_GD_MAX.In := IN_GT.tPr_GT_Gas.Ai;
		xGR_MAX_FA_GD_MAX.Gw := Para.rPr_GT_LimMax;
		xGR_MAX_FA_GD_MAX.Hy := Para.rPr_GT_HyMax;
		xGR_MAX_FA_GD_MAX();

		xTON_FA_T_GD_MAX.IN := IN_GT.tPB2MM.bParaSetupOk AND xGR_MAX_FA_GD_MAX.Q;
		xTON_FA_T_GD_MAX.PT := T#2s;
		xTON_FA_T_GD_MAX();

		GD_MAX := GD_MAX_a AND xTON_FA_T_GD_MAX.Q;
	ELSE
		MS_GD	 := FALSE;
		GD_MIN	 := FALSE;
		GD_MIN_W := FALSE;
		GD_MAX	 := FALSE;
		OUT_GT.rP_Red_GasPr_Norm := 1.0;
	END_IF;

	(* Tecjet differential pressure *)
	IF (Para.iTJ_DPress_PowRed_Mode = 1 OR Para.iTJ_DPress_PowRed_Mode = 2) AND IN_GT.rP_Act_Norm_Filt >= 0.4 AND IN_GT.iN_GMU_Devices <> 0 AND Para.bTJ_Exist THEN
		rGMU_Pr_DiffGas_min := 1.00;

		FOR i := 1 TO IN_GT.iN_GMU_Devices BY 1 DO					(* select the minimum delta P of all Tecjet valves *)
			IF rGMU_Pr_DiffGas_min > IN_GT.rGMU_Pr_DiffGas[i] AND IN_GT.rGMU_Pos_Valve_Prom[i] > 0.005 THEN
					rGMU_Pr_DiffGas_min := IN_GT.rGMU_Pr_DiffGas[i];
			END_IF;
		END_FOR
		xTON_TJdeltaP_min(IN := rGMU_Pr_DiffGas_min < Para.rTJ_DPress_Min, PT := Para.tiTJ_DPress_Min_Delay);
		bPr_TecJetDP_Min	   	:= 	xTON_TJdeltaP_min.Q;		(* stop the motor with priority 3 *)
	ELSE
		xTON_TJdeltaP_min(IN  := FALSE, PT :=  Para.tiTJ_DPress_Min_Delay);
		bPr_TecJetDP_Min 		:= FALSE;
	END_IF;

	IF 	Para.iTJ_DPress_PowRed_Mode = 2 AND IN_GT.rP_Act_Norm_Filt >= 0.4 AND IN_GT.iN_GMU_Devices <> 0 AND Para.bTJ_Exist THEN (* Gas supply pressure measurement activated and function of power reduction based on delta P of Tecjet activated*)
		SimPID_deltaP_TJ.ssMethodType		:=	3;							 (* Controller Mode 3 --> Automatic mode *)
		SimPID_deltaP_TJ.w					:=  Para.rTJ_DPress_P_Red_Start; (* 0.02bar is the mimimum for this parameter *)
		SimPID_deltaP_TJ.x					:=	rGMU_Pr_DiffGas_min;
		SimPID_deltaP_TJ.P 					:=  Para.rCtr_TJ_DPress_kp;
		SimPID_deltaP_TJ.I 					:=  Para.rCtr_TJ_DPress_ki;
		SimPID_deltaP_TJ.umin       		:=  MAX(IN_GT.rP_Set_Min_Norm, 0.4) - LIMIT(MAX(IN_GT.rP_Set_Min_Norm, 0.4), IN_GT.rP_Set_Unred_Norm, 1);

		SimPID_deltaP_TJ();

		IF SimPID_deltaP_TJ.u < 0 THEN
			OUT_GT.rP_Red_TJDiffPr_Norm := LIMIT(MAX(IN_GT.rP_Set_Min_Norm, 0.4), SimPID_deltaP_TJ.u + rP_Set_Unred_Norm_GT, 1); //Start reduction from actual power
			bPr_TecJetDP_P_Red := TRUE;
		ELSE
			OUT_GT.rP_Red_TJDiffPr_Norm := 1;
			rP_Set_Unred_Norm_GT := IN_GT.rP_Set_Unred_Norm;
			bPr_TecJetDP_P_Red := FALSE;
		END_IF;
	ELSE
		OUT_GT.rP_Red_TJDiffPr_Norm := 1;
		bPr_TecJetDP_P_Red := FALSE;
	END_IF;
	(************************************************************************************************************)
	(* Suction pressure *)
	IF Para.bP_GT_SuctPrActive THEN
		(* Suction pressure measurement signal failure *)
		MS_SD := IN_GT.tPB2MM.bParaSetupOk AND NOT IN_GT.tPr_GT_Suct.GoodQual;

		(* Reduction due to Suction pressure *)
		RED_SD_a := Para.bP_Red_SuctPrActive AND NOT MS_SD AND NOT IN_GT.tP_Red_SuctPrActive.Di AND IN_GT.tPB2MM.bParaSetupOk;
		xSigScalR_FA_SD_RED.X  := IN_GT.tPr_GT_Suct.Ai;
		xSigScalR_FA_SD_RED.X1 := Para.rP_Red_SuctPrStart;
		xSigScalR_FA_SD_RED.Y1 := 1.00;
		xSigScalR_FA_SD_RED.X2 := Para.rP_Red_SuctPrHalfLoad;
		xSigScalR_FA_SD_RED.Y2 := 0.50;
		xSigScalR_FA_SD_RED();
		IF RED_SD_a THEN
			OUT_GT.rP_Red_SuctPr_Norm := LIMIT(0,xSigScalR_FA_SD_RED.Y_SCAL,1.00);
		ELSE
			OUT_GT.rP_Red_SuctPr_Norm := 1.0;
		END_IF;

		(* Suction pressure minimum *)
		xGR_MINR_FA_SDMIN.In := ABS(IN_GT.tPr_GT_Suct.Ai);
		xGR_MINR_FA_SDMIN.Hy := Para.rPr_GT_SuctPrHyMin;
		xGR_MINR_FA_SDMIN.Gw := ABS(Para.rPr_GT_SuctPrLimMin);
		xGR_MINR_FA_SDMIN();
		xTON_FA_T_SD_MIN.IN  := xGR_MINR_FA_SDMIN.Q AND IN_GT.tPB2MM.bParaSetupOk;
		xTON_FA_T_SD_MIN.PT  := T#2s;
		xTON_FA_T_SD_MIN();
		bMsgDummy_Min_SuctPr := xTON_FA_T_SD_MIN.Q;	// formerly SD_MIN

		(* Suction pressure maximum *)
		xGR_MAXR_FA_SDMAX.In := ABS(IN_GT.tPr_GT_Suct.Ai);
		xGR_MAXR_FA_SDMAX.Hy := Para.rPr_GT_SuctPrHyMax;
		xGR_MAXR_FA_SDMAX.Gw := ABS(Para.rPr_GT_SuctPrLimMax);
		xGR_MAXR_FA_SDMAX();
		xTON_FA_T_SD_MAX.IN  := xGR_MAXR_FA_SDMAX.Q AND IN_GT.tPB2MM.bParaSetupOk;
		xTON_FA_T_SD_MAX.PT  := T#2s;
		xTON_FA_T_SD_MAX();
		bMsgDummy_Max_SuctPr := xTON_FA_T_SD_MAX.Q;  // formerly SD_MAX
	ELSE
		MS_SD 				 := FALSE;
		bMsgDummy_Min_SuctPr := FALSE;
		bMsgDummy_Max_SuctPr := FALSE;
		OUT_GT.rP_Red_SuctPr_Norm := 1.0;
	END_IF;

	(************************************************************************************************************)
	(* O2_MAX A1087 O2 content high *)
	IF Para.bGT_O2Active THEN
		(* O2 content measurement signal error *)
		MS_O2   := IN_GT.tPB2MM.bParaSetupOk AND NOT IN_GT.tGT_O2.GoodQual;
		MS_O2_W := IN_GT.tPB2MM.bParaSetupOk AND NOT IN_GT.tGT_O2.GoodQual AND NOT Para.bGT_O2MaxTripActive;
		MS_O2_A := IN_GT.tPB2MM.bParaSetupOk AND NOT IN_GT.tGT_O2.GoodQual AND Para.bGT_O2MaxTripActive;

		(* O2 content maximum  *)
		xGR_MAX_FA_O2_MAX.In := IN_GT.tGT_O2.Ai;
		xGR_MAX_FA_O2_MAX.Hy := Para.rGT_O2HyMax;
		xGR_MAX_FA_O2_MAX.Gw := Para.rGT_O2LimMax;
		xGR_MAX_FA_O2_MAX();
		xTON_FA_T_O2_MAX.IN := xGR_MAX_FA_O2_MAX.Q AND IN_GT.tPB2MM.bParaSetupOk;
		xTON_FA_T_O2_MAX.PT := T#2s;
		xTON_FA_T_O2_MAX();
		O2_MAX := xTON_FA_T_O2_MAX.Q AND Para.bGT_O2MaxTripActive;
	ELSE
		MS_O2	:= FALSE;
		MS_O2_W := FALSE;
		MS_O2_A := FALSE;
		O2_MAX  := FALSE;
	END_IF;

	(************************************************************************************************************)
	(* Gas temperature L089 *)
	IF Para.bT_GT_Active THEN

		(* Gas temperature measurement signal error *)
		MS_GT  := IN_GT.tPB2MM.bParaSetupOk AND NOT IN_GT.tT_GT.GoodQual;

		(* Gas temperature minimum *)
		xGR_MIN_FA_GT_MIN.In := IN_GT.tT_GT.Ai;
		xGR_MIN_FA_GT_MIN.Hy := Para.rT_GT_HyMin;
		xGR_MIN_FA_GT_MIN.Gw := Para.rT_GT_LimMin;
		xGR_MIN_FA_GT_MIN();
		xTON_FA_T_GT_MIN.IN := IN_GT.tPB2MM.bParaSetupOk AND xGR_MIN_FA_GT_MIN.Q;
		xTON_FA_T_GT_MIN.PT := T#2s;
		xTON_FA_T_GT_MIN();
		GT_MIN := xTON_FA_T_GT_MIN.Q;

		(* Gas temperature maximum *)
		xGR_MAX_FA_GT_MAX.In := IN_GT.tT_GT.Ai;
		xGR_MAX_FA_GT_MAX.Hy := Para.rT_GT_HyMax;
		xGR_MAX_FA_GT_MAX.Gw := Para.rT_GT_LimMax;
		xGR_MAX_FA_GT_MAX();
		xTON_FA_T_GT_MAX.IN := IN_GT.tPB2MM.bParaSetupOk AND xGR_MAX_FA_GT_MAX.Q;
		xTON_FA_T_GT_MAX.PT := T#2s;
		xTON_FA_T_GT_MAX();
		GT_MAX := xTON_FA_T_GT_MAX.Q;
	ELSE
		MS_GT 	:= FALSE;
		GT_MIN	:= FALSE;
		GT_MAX	:= FALSE;
	END_IF;

	(************************************************************************************************************)
	(* Gas quantity  L105 *)
	IF Para.bVol_GT_Active THEN
		MS_GM := IN_GT.tPB2MM.bParaSetupOk AND NOT IN_GT.tVol_GT.GoodQual;
	ELSE
		MS_GM := FALSE;
	END_IF;

	(************************************************************************************************************)
	(* Freigabe aus Gasstation (W3153) *)
	IF IN_GT.bRelGasPlant_Bus_Active THEN
		xTOF_FA_T_FG_GAS.IN := IN_GT.bRelGasPlant_Bus;
	ELSE
		xTOF_FA_T_FG_GAS.IN := IN_GT.tRelGasPlant.Di;
	END_IF;

	xTOF_FA_T_FG_GAS.PT := T#2s;
	xTOF_FA_T_FG_GAS();
	T_FG_GAS := xTOF_FA_T_FG_GAS.Q;

	xTP_FA_FG_GAS.IN := ((IN_GT.bEng_Aux_Dem OR NOT FGGAS) AND NOT OUT_GT.bGT2_Select) AND NOT T_FG_GAS;
	IF bTestEnabled THEN
		xTP_FA_FG_GAS.PT := T#3s;
	ELSE
		xTP_FA_FG_GAS.PT := T#300s;
	END_IF;
	xTP_FA_FG_GAS();
	FGGAS := NOT ((IN_GT.bEng_Aux_Dem OR NOT FGGAS) AND NOT OUT_GT.bGT2_Select AND
	(xTP_FA_FG_GAS.Q OR NOT T_FG_GAS));

	(* 	Blockierung Modul (pb7/M_BLOCK)  *)
	OUT_GT.bGasSupplyOk := OUT_GT.bGT2_Select OR (NOT CH4_MIN_W AND NOT MM2VIS.bMsg_Dummy_Warn_CV AND NOT GD_MIN_W AND FGGAS);

	(************************************************************************************************************)
	(* Alarms *)
	(* 1028 gas pressure low gas train 1 *)
	xTON_GDMI1(IN := (NOT IN_GT.tPr_GT1_Min.Di OR NOT IN_GT.tPr_GT1_1_Min.Di OR IN_GT.bPr_GT1_Min_Cust), PT := T#2s);
	HM_GDMI1 := xTON_GDMI1.Q;

	ZM_GDMI1 := ((HM_GDMI1 AND NOT Para.bPurgecycle_Active) OR ((NOT IN_GT.tPr_GT1_Min.Di OR NOT IN_GT.tPr_GT1_1_Min.Di OR IN_GT.bPr_GT1_Min_Cust) AND Para.bPurgecycle_Active)) AND
	(FG_GDRUW OR (ZM_GDMI1 AND NOT Para.bGCActive)) AND
	NOT OUT_GT.bGT2_Select AND
	(T_GDRUW OR NOT Para.bGCActive);

	bMsg1028_Set := (ZM_GDMI1 AND NOT Para.bVISA) OR (HM_GDMI1 AND Para.bVISA);

	(* 1030 Gas pressure low gas train 2 *)
	xTON_GDMI2(IN := NOT IN_GT.tPr_GT2_Min.Di, PT := T#2s);
	HM_GDMI2 := xTON_GDMI2.Q;

	ZM_GDMI2 := ((HM_GDMI2 AND NOT Para.bPurgecycle_Active) OR (NOT IN_GT.tPr_GT2_Min.Di AND Para.bPurgecycle_Active)) AND
	(FG_GDRUW OR ZM_GDMI2) AND (OUT_GT.bGT2_Select OR UW_GST2);

	bMsg1030_Set := (ZM_GDMI2 AND NOT Para.bVISA)  OR (HM_GDMI2 AND Para.bVISA);

	(* 1057 gas train 1 gas pressure high *)
	(* flag for deactivating gas pressure monitoring (V1.70.1) *)
	xTOF_N2_GASV(IN:= IN_GT.tN2_ScavGV_CoOpen.Do, PT := T#5s);		// before realised in N2spueleung #41
	T_N2_GASV := xTOF_N2_GASV.Q;

	xTON_GDMA1.IN := (NOT T_N2_GASV OR NOT IN_GT.bRel_ScavN2) AND (NOT IN_GT.tPr_GT1_Max.Di OR NOT IN_GT.tPr_GT1_1_Max.Di OR IN_GT.bPr_GT1_Max_Cust);
	xTON_GDMA1.PT := T#4s;
	xTON_GDMA1();

	ZM_GDMA1 := IN_GT.tEng_Run.Do AND M_GASV1 AND
	((Para.bPurgecycle_Active AND xTON_GDMA1.IN AND FG_GDRUW) OR
	(NOT Para.bPurgecycle_Active AND xTON_GDMA1.Q));

	xTON_GDMA1_VISA.IN := (NOT IN_GT.tPr_GT1_Max.Di OR NOT IN_GT.tPr_GT1_1_Max.Di OR IN_GT.bPr_GT1_Max_Cust);
	xTON_GDMA1_VISA.PT := T#3s;
	xTON_GDMA1_VISA();

	bMsg1057_Set := (ZM_GDMA1 AND NOT Para.bVISA) OR (xTON_GDMA1_VISA.Q AND Para.bVISA);

	(* 1058 gas pressure high gas train 2 *)
	xTON_GDMA2.IN := (NOT T_N2_GASV OR NOT IN_GT.bRel_ScavN2) AND NOT IN_GT.tPr_GT2_Max.Di;
	xTON_GDMA2.PT := T#4s;
	xTON_GDMA2();

	ZM_GDMA2 := IN_GT.tEng_Run.Do AND M_GASV2 AND
	((NOT Para.bPurgecycle_Active AND xTON_GDMA2.Q) OR
	(Para.bPurgecycle_Active AND xTON_GDMA2.IN AND FG_GDRUW));

	xTON_GDMA2_VISA.IN := NOT IN_GT.tPr_GT2_Max.Di;
	xTON_GDMA2_VISA.PT := T#3s;
	xTON_GDMA2_VISA();

	bMsg1058_Set := (ZM_GDMA2 AND NOT Para.bVISA) OR (xTON_GDMA2_VISA.Q AND Para.bVISA);

	(* 3353 gas pressure low gas train 1 - line 2 *)
	xTON_GDMI1_2(IN := NOT IN_GT.tPr_GT1_2_Min.Di, PT := T#2s);
	HM_GDMI1_2 	:= AKT_Gastrecke1_2 AND xTON_GDMI1_2.Q;

	ZM_GDMI1_2 	:= 	((xTON_GDMI1_2.Q AND NOT Para.bPurgecycle_Active) OR (NOT IN_GT.tPr_GT1_2_Min.Di AND Para.bPurgecycle_Active)) AND
	(FG_GDRUW OR (ZM_GDMI1_2 AND NOT Para.bGCActive)) AND
	NOT OUT_GT.bGT2_Select AND
	(T_GDRUW OR NOT Para.bGCActive);

	bMsg3353_Set :=	AKT_Gastrecke1_2 AND
	((ZM_GDMI1_2 AND NOT Para.bVISA) OR (xTON_GDMI1_2.Q AND Para.bVISA));

	(* 3354 gas pressure low gas train 1 - line 3 *)
	xTON_GDMI1_3(IN := NOT IN_GT.tPr_GT1_3_Min.Di, PT := T#2s);
	HM_GDMI1_3 	:= AKT_Gastrecke1_3 AND xTON_GDMI1_3.Q;

	ZM_GDMI1_3 	:= 	((xTON_GDMI1_3.Q AND NOT Para.bPurgecycle_Active) OR (NOT IN_GT.tPr_GT1_3_Min.Di AND Para.bPurgecycle_Active)) AND
	(FG_GDRUW OR (ZM_GDMI1_3 AND NOT Para.bGCActive)) AND
	NOT OUT_GT.bGT2_Select AND
	(T_GDRUW OR NOT Para.bGCActive);

	bMsg3354_Set :=	AKT_Gastrecke1_3 AND
	((ZM_GDMI1_3 AND NOT Para.bVISA) OR (xTON_GDMI1_3.Q AND Para.bVISA));

	(* 3355 gas pressure low gas train 1 - line 4 *)
	xTON_GDMI1_4(IN := NOT IN_GT.tPr_GT1_4_Min.Di, PT := T#2s);
	HM_GDMI1_4 	:= AKT_Gastrecke1_4 AND xTON_GDMI1_4.Q;

	ZM_GDMI1_4 	:= 	((xTON_GDMI1_4.Q AND NOT Para.bPurgecycle_Active) OR (NOT IN_GT.tPr_GT1_4_Min.Di AND Para.bPurgecycle_Active)) AND
	(FG_GDRUW OR (ZM_GDMI1_4 AND NOT Para.bGCActive)) AND
	NOT OUT_GT.bGT2_Select AND
	(T_GDRUW OR NOT Para.bGCActive);

	bMsg3355_Set :=	AKT_Gastrecke1_4 AND
	((ZM_GDMI1_4 AND NOT Para.bVISA) OR (xTON_GDMI1_4.Q AND Para.bVISA));

	(* 3356 gas train 1 gas pressure high - line 2 *)
	xTON_GDMIA1_2(IN := (NOT T_N2_GASV OR NOT IN_GT.bRel_ScavN2) AND NOT IN_GT.tPr_GT1_2_Max.Di, PT := T#4s);
	ZM_GDMA1_2	:= ((NOT Para.bPurgecycle_Active AND xTON_GDMIA1_2.Q) OR
	(Para.bPurgecycle_Active AND xTON_GDMIA1_2.IN AND FG_GDRUW)) AND
	M_GASV1 AND IN_GT.tEng_Run.Do;

	xTON_GDMA1_2_VISA(IN := NOT IN_GT.tPr_GT1_2_Max.Di, PT := T#3s);
	bMsg3356_Set := AKT_Gastrecke1_2 AND
	(ZM_GDMA1_2 AND NOT Para.bVISA) OR (xTON_GDMA1_2_VISA.Q AND Para.bVISA);

	(* 3357 gas train 1 gas pressure high - line 3 *)
	xTON_GDMIA1_3(IN := (NOT T_N2_GASV OR NOT IN_GT.bRel_ScavN2) AND NOT IN_GT.tPr_GT1_3_Max.Di, PT := T#4s);
	ZM_GDMA1_3 	:= ((NOT Para.bPurgecycle_Active AND xTON_GDMIA1_3.Q) OR
	(Para.bPurgecycle_Active AND xTON_GDMIA1_3.IN AND FG_GDRUW)) AND
	M_GASV1 AND IN_GT.tEng_Run.Do;

	xTON_GDMA1_3_VISA(IN := NOT IN_GT.tPr_GT1_3_Max.Di, PT := T#3s);
	bMsg3357_Set := AKT_Gastrecke1_3 AND
	(ZM_GDMA1_3 AND NOT Para.bVISA) OR (xTON_GDMA1_3_VISA.Q AND Para.bVISA);

	(* 3358 gas train 1 gas pressure high - line 4 *)
	xTON_GDMIA1_4(IN := (NOT T_N2_GASV OR NOT IN_GT.bRel_ScavN2) AND NOT IN_GT.tPr_GT1_4_Max.Di, PT := T#4s);
	ZM_GDMA1_4 	:= ((NOT Para.bPurgecycle_Active AND xTON_GDMIA1_4.Q) OR
	(Para.bPurgecycle_Active AND xTON_GDMIA1_4.IN AND FG_GDRUW)) AND
	M_GASV1 AND IN_GT.tEng_Run.Do;

	xTON_GDMA1_4_VISA(IN := NOT IN_GT.tPr_GT1_4_Max.Di, PT := T#3s);
	bMsg3358_Set := AKT_Gastrecke1_4 AND
	(ZM_GDMA1_4 AND NOT Para.bVISA) OR (xTON_GDMA1_4_VISA.Q AND Para.bVISA);

	(* 9371 Measuring signal failure setpoint - Gas mixing *)
	IF IN_GT.tGT_RatioMix_Set.Exist AND NOT IN_GT.tGT_RatioMix_Set.GoodQual THEN
		bMsg9371_Set := TRUE;
	ELSE
		bMsg9371_Set := FALSE;
	END_IF;

END_PROGRAM
```

#### spec_gas.var - Local variables
```iecst
VAR
	CH4_MIN : BOOL := 0; (* CH4-Gehalt minimum *)
	CH4_MIN_W_1 : BOOL;
	CH4_MIN_W_a : BOOL;
	CV_MIN : BOOL := 0; (* Heizwert minimum *)
	CV_MIN_W_a : BOOL;
	GD_MAX_a : BOOL;
	GD_MIN : BOOL;
	GD_MIN_a : BOOL;
	GD_MIN_W : BOOL;
	RED_CH4_a : BOOL;
	RED_CV_a : BOOL;
	RED_GD_a : BOOL;
	RED_SD_a : BOOL;
	S_MS_CH4 : BOOL := 0; (* Messignal CH4-Gehalt *)
	S_MS_CV : BOOL := 0; (* Messignal Heizwert *)
	T_FG_GAS : BOOL;
	xGR_MAXR_FA_SDMAX : GR_MAXR;
	xGR_MAX_FA_GD_MAX : GR_MAXR;
	xGR_MAX_FA_GT_MAX : GR_MAXR;
	xGR_MAX_FA_O2_MAX : GR_MAXR;
	xGR_MINR_FA_CH4_MIN_A : GR_MINR;
	xGR_MINR_FA_CH4_MIN_W : GR_MINR;
	xGR_MINR_FA_CV_MIN_A : GR_MINR;
	xGR_MINR_FA_CV_MIN_W : GR_MINR;
	xGR_MINR_FA_SDMIN : GR_MINR;
	xGR_MIN_FA_GD_MIN : GR_MINR;
	xGR_MIN_FA_GT_MIN : GR_MINR;
	xSigScalR_FA_CH4_GMV : xSigScal_R;
	xSigScalR_FA_CH4_RED : xSigScal_R;
	xSigScalR_FA_GD_RED : xSigScal_R;
	xSigScalR_FA_SD_RED : xSigScal_R;
	xSigScal_FA_CV_RED : xSigScal_R;
	xSigScal_R_FA_CalVal_GMV : xSigScal_R;
	xTOF_FA_T_FG_GAS : TOF;
	xTOF_N2_GASV : TOF;
	xTON_FA_CH4_MIN : TON;
	xTON_FA_CV_MIN : TON;
	xTON_FA_T_CH4_A : TON;
	xTON_FA_T_CH4_W : TON;
	xTON_FA_T_CV_A : TON;
	xTON_FA_T_CV_W : TON;
	xTON_FA_T_GD_MAX : TON;
	xTON_FA_T_GT_MAX : TON;
	xTON_FA_T_GT_MIN : TON;
	xTON_FA_T_O2_MAX : TON;
	xTON_FA_T_SD_MAX : TON;
	xTON_FA_T_SD_MIN : TON;
	xTON_GDMA1 : TON;
	xTON_GDMA1_2_VISA : TON;
	xTON_GDMA1_3_VISA : TON;
	xTON_GDMA1_4_VISA : TON;
	xTON_GDMA1_VISA : TON;
	xTON_GDMA2 : TON;
	xTON_GDMA2_VISA : TON;
	xTON_GDMI1 : TON;
	xTON_GDMI1_2 : TON;
	xTON_GDMI1_3 : TON;
	xTON_GDMI1_4 : TON;
	xTON_GDMI2 : TON;
	xTON_GDMIA1_2 : TON;
	xTON_GDMIA1_3 : TON;
	xTON_GDMIA1_4 : TON;
	xTP_FA_FG_GAS : TP;
	xTP_FA_GD_MIN_W : TP;
	Y_SCAL_CalVal : REAL;
	ZM : BOOL := 0; (* Zwischenmerker *)
	ZM_GDMA1_2 : BOOL;
	ZM_GDMA1_3 : BOOL;
	ZM_GDMA1_4 : BOOL;
	ZM_GDMI1_2 : BOOL;
	ZM_GDMI1_3 : BOOL;
	ZM_GDMI1_4 : BOOL;
	i : INT;
	SimPID_deltaP_TJ : SimPID4 := (0);
	rGMU_Pr_DiffGas_min : REAL; (* Minimum gas proportional valve differential pressure *)
	xTON_TJdeltaP_min : TON;
	rReductionPowerH2 : REAL; (* Power reduction value [%Pnom] *)
	rReductionPowerH2_MSF : REAL; (* Power reduction value [%Pnom] *)
	xGR_MAXR_H2_Comp : GR_MAXR;
	rGwH2_Comp : REAL := 0.02; (* Trehshold of H2 content [%] *)
	rHyH2_Comp : REAL := 0.01; (* Trehshold of H2 content [%] *)
	xGR_MAXR_FA_H2_MAX_A : GR_MAXR;
	xGR_MAXR_FA_H2_MAX_W : GR_MAXR;
END_VAR
```

### Program Logical/Gastrain/gas_zust (IEC) - Gas_zust

#### gas_zustCyclic.st - Cyclic code
```iecst
(* BERECHNUNG GAS-ZUSTANDSZAHL
....................._
VER	Datum/Name	Änderung
V172	27.06.02/LH	erstellt
 	    17.09.02/LH	korrigiert für AS 2.2
V190	18.06.04/LH	Vermeidung von Rundungsfehlern
V2201	08.08.07/LH	Pakistan-Standard: Normaltemp. = 15°C
 			        Anbindung an "spec_gas"-Werte
V3.99	21-09-2013	Ganguly/Denk, generated for modular software*)

PROGRAM _CYCLIC

    (* Filtering turbo boost pressure *)
	xLCRPT1_PressP2.x := IN_GT.rPr_Ch_P2s_Avg_UF;
	xLCRPT1_PressP2();
	pl_ist := xLCRPT1_PressP2.y;

	(* Determining the normal temperature for conversion *)
	IF (Para.iCountry = iPakistan) THEN
		Tn_ls := 288.15;
	ELSE
		Tn_ls := Tn;   // Tn = 273.15 K is stored as a constant
	END_IF;

	(* Operating temperature 0.01°K => Temperature in Kelvin = Temperature in Celsius + (273.15 OR 288.15) *)
	(* Calculating  the temperature relation *)
	VT := Tn_ls/(IN_GT.tT_GT.Ai + Tn);

	(*-----------------------------------------------------------*)
	(* Detecting the air pressure *)
	IF NOT IN_GT.bEng_Aux_Dem_CDR THEN
	    (* Air pressure *)
		p_luft := pl_ist;
	ELSE
	    (* Actual boost pressure *)
		p_luft := p_luft;
	END_IF;

	(* Assigning Gas pressure depending on whether absolute gas pressure measurement is active or not *)
	IF NOT Para.bPr_GasPrAbsActive THEN
		GAS_PB := p_luft + IN_GT.tPr_GT_Gas.Ai ;
	ELSE
		GAS_PB := 0.0 + IN_GT.tPr_GT_Gas.Ai ;
	END_IF;

	(* Calculation of the pressure relation *)
	Vp := GAS_PB/pn;

	(*-----------------------------------------------------------*)
	(* Berechnung Zustandzahl (ZSZ(x1000)=(Vt*Vp)/1000°K) *)
	(* Calculation Gas volume correction factor K = adjustment factor = ( 1/gas law deviation factor) *)
	ZSZ := VT * Vp * K;

END_PROGRAM
```

#### gas_zustInit.st
```iecst
PROGRAM _INIT

(* Initialization for low pass filter initialization *)
xLCRPT1_PressP2.enable := TRUE;
xLCRPT1_PressP2.t      := 1;
xLCRPT1_PressP2.set    := FALSE;

END_PROGRAM
```

#### gas_zust.var - Local variables
```iecst
(********************************************************************
 * COPYRIGHT -- INNIO Company
 ********************************************************************
 * Program: gas_zust
 * File: gas_zust.var
 * Author: 105051626
 * Created: April 19, 2012
 ********************************************************************
 * Local variables of program gas_zust
 ********************************************************************)
VAR

	Tn_ls : REAL; (* Normgastemperatur länderspezifisch *)
	VT : REAL; (* Temperaturverhältnis *)
END_VAR
VAR CONSTANT
	Tn : REAL := 273.15; (*Normal temperature*)
END_VAR
VAR
	p_luft : REAL := 1.013; (*Air pressure [Bar]*)
	GAS_PB : REAL; (*Operating gas pressure*)

	Vp : REAL; (* Druckverhältnis *)
	xLCRPT1_PressP2 : LCRPT1;
END_VAR
VAR CONSTANT
	iPakistan : INT := 92; (*country code, TEMP Solution!!!*)
END_VAR
```

### Program Logical/Gastrain/gasum_st (IEC) - gasum_st

#### gasum_stCyclic.st - Cyclic code
```iecst
(* GASUMSCHALTUNG IM STILLSTAND

VER	Datum/Name	Änderung
V170	04.04.02/LH	erstellt
V2071	15.02.05/LH	angepasst für Gasstrecke 2 = Gasart 3
 		03.03.05/LH	neue Variable "OUT_GT.bGT_TypSwhActiveHalt" eingeführt
V220	19.02.07/LH	angepasst für X20-Einführung
V2.60.0	06.10.2009  Lettenb		task activation added
V03.99.00.00	21.09.2013	Denk		generated for modular software
				28.05.2013	lettenb.	bTestEnabled Para -> loc.var
V04.01.00.00	31.07.2014  Denk		Para.bGT_MixActiveEngStop added

Instructions for use:
------------------------------
activate task if used
set connections acc. comment *)

PROGRAM _CYCLIC

(* task activation *)
IF NOT Para.bGT_MixActiveEngStop THEN
	RETURN;
END_IF;

	(* Anzahl der Gasstrecken > 1 *)
	(* Number of Gas trains > 1 *)
	OUT_GT.bGT_TypSwhActiveHalt := TRUE;

	(* Anzahl der Gasarten > 2 *)
	(* Number of Gas type > 2 *)
	ZM  := Para.iIdx_Gastyp > 2;

	(* Rückschaltung *)
	(* ????? code revision *)
	ST6 := (OUT_GT.bSelGasTypAut OR NOT OUT_GT.bSelGasTyp3) AND (NOT IN_GT.tGT_TypSwitch.Di OR NOT OUT_GT.bSelGasTypAut) AND AF_GASUM;

	IF bTestEnabled THEN xTON_FA_T6.PT:= T#5s;
	ELSE				 xTON_FA_T6.PT:= T#5m;
	END_IF;
	xTON_FA_T6(IN:= ST6);
	AT6 := ST6 AND (NOT OUT_GT.bGV_On OR xTON_FA_T6.Q);

	(* Anforderung Gasumschaltung *)
	(* Demand Gas switch *)
	AF_GASUM := ((OUT_GT.bSelGasTypAut AND (IN_GT.tGT_TypSwitch.Di OR AF_GASUM)) OR OUT_GT.bSelGasTyp3) AND NOT AT6 AND ZM;

	(* Anwahl Gasstrecke 2 *)
	(* Select Gas train 2 *)
	OUT_GT.bGT2_Select := (AF_GASUM AND NOT IN_GT.bEng_Dem_Bloc) OR (OUT_GT.bGT2_Select AND
	                      (IN_GT.bEng_Dem_Bloc OR AF_GASUM));

	(* Anforderung Entlastung fur Gasumschaltung *)
	(* Demand unloading for Gas train switch *)
	OUT_GT.bGT_DemRelGasTypSwh := (NOT OUT_GT.bGT2_Select AND AF_GASUM) OR (OUT_GT.bGT2_Select AND NOT AF_GASUM);

	(* Gasventile *)
	(* Gas valves *)
	M_GASV1 := NOT OUT_GT.bGT2_Select;
	M_GASV2 := OUT_GT.bGT2_Select;

END_PROGRAM
```

#### gasum_st.var - Local variables
```iecst
(********************************************************************
 * COPYRIGHT -- INNIO Company
 ********************************************************************
 * Program: gasum_st
 * File: gasum_st.var
 * Author: 105051626
 * Created: April 19, 2012
 ********************************************************************
 * Local variables of program gasum_st
 ********************************************************************)
VAR
	ZM : BOOL := 0; (* Zwischenmerker*)
	ST6 : BOOL;
	AF_GASUM : BOOL; (* Anforderung Gasumschaltung *)
	xTON_FA_T6 : TON;
	AT6 : BOOL;
END_VAR
```

### Program Logical/Gastrain/pb5 (IEC) - pb5

#### pb5Cyclic.st - Cyclic code
```iecst
(********************************************************************************
pb5 			gas train testing

This code is confidential and proprietary to the INNIO Company.
It may not be used in any form, or reproduced in any manner,
without written permission of the INNIO Company.
Copyright, INNIO Company, 2025

Customized modifications: -
------------------------

History:
-------
V0.1	06.07.98/Pa	erstellt
 	    24.11.98/Pa	korrekturlesung
V2071	07.07.05/LH	Prüfzeiten für DK2F angepasst
    	03.03.05/LH	Anzahl Gasstrecken < 2
V220	19.02.07/LH	angepasst für X20-Einführung
V3.20.0	04.11.2010  lettenb.	Para.bPurgecycle_Active added (test gas train before start)
V03.99.00	21.09.2013	Ganguly 	generated for modular software
V03.99.01	20.02.2013	Denk		V3.30 changes inserted
			22.11.2013	lettenb.	V3.50 test gas train with exh.gas scavenging added
			20.02.2014	lettenb.	bugfix gas train check for BR2,3,4
V04.01.00	15.07.2014	Denk		bugfix M_STGAS1
			12.09.2014	lettenb.	M_DREHZ added(purge cycle: to avoid tight check during eng.operation)
V04.03.00	05.10.2015	Denk		Prechamber gas train safety device
			01.06.2016  lettenb.	xTP_TP_vorStart2 added for BR234 with purgecycle, bugfix
V04.04.00	13.10.2016	Denk		bMsg1027 setting function when remote reset
V04.06.00	25.06.2018	Perktold	IN_GT.bGT_Check4FastStart, OUT_GT.bGT2_SafeDevOK and OUT_GT.bPCGT_SafeDevOK implemented
V04.07.00 	24.09.2018	Denk		Avoid second start of gas safety device (DPFR-20180821-0202)
V04.07.01 	04.04.2019	Zengerer	requisition variants selection: chapter 5-configuration gas leakage MGV, LIMIT(T#600ms, Para.tiGT_TestDuration
V04.09.00	25.10.2019	Zengerer	release option 4 MEGAGas- Demand compressor option
			26.11.2019	Zengerer	xF_trig_GK, xR_trig_PO removed for better readability, NO functional change
			16.01.2020	Zengerer	release option 4 MEGAGas- delayed valve check demand bDelay_GDKG_GCStarting, option 1 and 2 covered with Megagas ELSE, OUT_GT.tGT1_SafeDevice.Do := (corr.Jan2020)
			05.03.2020	Denk		Testing time gas train 1 and 2 increased to 130 sec. Mandatory for new MegaGas valves function
V04.14.00	23.02.2025	Tinello		Gas leakage check moved to SafetyPLC
V04.25.00	30.12.2025	Tinello		Logic modified because of SafetyPLC

Instructions for use:
--------------------

Outstandings:
------------
Para.iGasTrain_Type  TODO: VALIDATION FOR OPTION 4, TO ALLOW PARA VALUE>2
********************************************************************************)

PROGRAM _CYCLIC

	Para.iGasTrain_Type := LIMIT(1 , Para.iGasTrain_Type, 4);	(* TODO: VALIDATION FOR OPTION 4, TO ALLOW PARA VALUE>2 *)
	Para.iGasTrain_Upstream_Type;								(* V4.07 new  *)

	(*Customisation Interface from Module Customized: *)
	IN_GT.tCU2GT.tiGT_TestDuration := LIMIT(T#1s , IN_GT.tCU2GT.tiGT_TestDuration, T#5m);		(* optional prepared customizable interface  *)
	IN_GT.tCU2GT.tiGCPulse_Duration_min;			(* optional prepared customizable interface  *)
	IN_GT.tCU2GT.tiGV_Feedback_Delay_max;			(* optional prepared customizable interface   *)
	IN_GT.tCU2GT.iGC_Select_Option ;				(* optional prepared customizable interface   *)
	IN_GT.tCU2GT.tiGV_Feedback_Delay_max := LIMIT(T#200ms , IN_GT.tCU2GT.tiGV_Feedback_Delay_max , T#240s);	(* optional prepared customizable interface  *)

	(* Acknowledgement Quiescent current loop OK *)
	xTON_FA_T94.IN := IN_GT.tSafetyLoop_Eng.Di;
	xTON_FA_T94.PT := T#5s;
	xTON_FA_T94();
	T94 := xTON_FA_T94.Q;

	(********************************************************************************************************************
	Safety-related application software source code: BEGIN
	Gas safety device must be triggered with Scavenging
	*********************************************************************************************************************)
	(* initiate gas train test *)
	xTOF_SafetyCheck_Run(IN:= EDGENEG(OUT_GT.tGT1_SafeDevice.Do), PT:= xTON_FA_T88.PT);
	xSR_GT_SafetyDevice2ndStartBlock(SET1 := EDGENEG(OUT_GT.tGT1_SafeDevice.Do), RESET := EDGENEG(IN_GT.bDemScavVa));

	(* initiate gas train test *)
	xTP_TP_vorStart.IN :=  (NOT M_DREHZ AND IN_GT.bDemScavVa AND NOT xSR_GT_SafetyDevice2ndStartBlock.Q1) OR (NOT M_DREHZ AND IN_GT.bGT_Check4FastStart AND (xTON_FA_T88.ET = xTON_FA_T88.PT OR xTON_FA_T88.ET = T#0s))
						OR (NOT M_DREHZ AND NOT Para.bEGScav_Active AND NOT xEngType.Type6 AND NOT xEngType.Type9);
	xTP_TP_vorStart.PT := T#1s;
	xTP_TP_vorStart();

	xTP_TP_vorStart2.IN := (NOT M_DREHZ AND Para.bPurgecycle_Active AND IN_GT.bEng_Dem); (* BR234 with purgecycle *)
	xTP_TP_vorStart2.PT := T#1s;
	xTP_TP_vorStart2();

	(* Gas train 1 test (DUNGS) *)
	xTP_FA_87.IN :=	NOT xTP_TP_vorStart.Q
				AND NOT xTP_TP_vorStart2.Q
				AND 	(T94 AND NOT MM2VIS.bMsg1027 AND NOT MM2VIS.bMsg3359 AND NOT MM2VIS.bMsg3360 AND NOT MM2VIS.bMsg3361)
				AND 	(bOMSS_MAT OR OUT_GT.bGT1_Check);
	xTP_FA_87.PT := T#1s;
	xTP_FA_87();
	T87 := xTP_FA_87.Q;

	IF Para.iGasTrain_Type = 1 THEN							(***option bit0 = '1' == STANDARD Gas Train (e.g. type Dungs)   ***)
		(*	option 1: no more special handling defined -> handled in ELSE from option 4	*)
	END_IF

	IF Para.iGasTrain_Type = 2 THEN 					  	(***option bit1 = '2'== Single Gas Valve Gas Train *)
		(*	option 2: no more special handling defined -> handled in ELSE from option 4	*)
	END_IF

		bMEGA_GasTrain :=  (Para.iGasTrain_Type = 4);	 	(***option bit2 = '4' == MEGA Gas Train, for wide pipe dimensions with 2 separate valves 	(V4.07	Requisition- supplied code parts included for MGV) *)
	IF 	bMEGA_GasTrain THEN  						 		(* bMEGA_GasTrain = Type = '4' == MEGA Gas Train , V4.07	 *)

		IN_GT.tCU2GT.tiGT_TestDuration;  							(*variable gas checking time parameter for bDelayForGascheck *)

		xTOF_RESET.IN := EDGEPOS(M_DREHZ);							(*TOF 5 sec extended 'engine in operation' trigger *)
		xTOF_RESET.PT := T#5s;
		xTOF_RESET();

		RS_GK.SET	 :=  EDGENEG(IN_GT.tAB2GT.bGnlTrip1  			(*memorize 'critical alarm' flag, triggered by critical alarm *)
							  OR IN_GT.tAB2GT.bGnlTrip2);
		RS_GK.RESET1 := M_DREHZ;
		RS_GK();

		xTOF_Shutdown.IN := EDGENEG(M_DREHZ);						(*TOF 2 sec after NOT 'engine in operation' trigger *)
		xTOF_Shutdown.PT := T#5s;
		xTOF_Shutdown();

		OUT_GT.tGT1_SafeDevice.Do := bDem_SafeDevice  AND (NOT bDelayGDKG_GCStarting);	(*(delayed) leakage check demand, to allow gas compressor generate sufficient pressure (corr.Jan2020)*)
		bDem_SafeDevice1 :=	(OUT_GT.tGT_GC_Dem.Do AND RS_GK.Q1) 	;					(*demand leakage check after critical alarm *)  //old Anf_GDKG is now ModuleGlobal, for task Biogas
		bDem_SafeDevice2 :=	(NOT T87 AND IN_GT.bEng_Aux_Dem_CDR) 	;					(*demand leakage check after normal engine operation *)
		bDem_SafeDevice3 :=	(IN_GT.tGT1_SafeDevOK.Di AND NOT xTOF_Shutdown.Q);			(*hold signal and surpress new leakage check at stopped engine after test ok *)
		bDem_SafeDevice	 :=	(bDem_SafeDevice1 OR bDem_SafeDevice2 OR bDem_SafeDevice3)
							AND NOT IN_GT.bSafetyPLC_Active;							(* SAFETY PLC *)

		xTON_GC_T100.IN := bDem_SafeDevice ;
		xTON_GC_T100.PT := LIMIT(T#600ms, IN_GT.tCU2GT.tiGT_TestDuration, T#240s);  	(*variable gas checking time parameter for bDelayForGascheck *)
		xTON_GC_T100();

		bDelayForGascheck := xTON_GC_T100.Q;
	ELSE

		OUT_GT.tGT1_SafeDevice.Do := NOT T87 AND NOT IN_GT.bSafetyPLC_Active;			(* SAFETY PLC *)

	END_IF
	(********************************************************************************************************************
	Safety-related application software source code: END
	Gas safety device must be triggered with Scavenging
	*********************************************************************************************************************)

	(* Testing time gas train 1 *)
	xTON_FA_T88.IN 	:=	OUT_GT.tGT1_SafeDevice.Do
						AND T94
						AND (bOMSS_MAT OR
							(OUT_GT.bGT1_Check AND NOT MM2VIS.bMsg1027 AND NOT MM2VIS.bMsg3359 AND NOT MM2VIS.bMsg3360 AND NOT MM2VIS.bMsg3361));

	IF bTestEnabled THEN		//for module test
		xTON_FA_T88.PT := T#1s;
	ELSE
		xTON_FA_T88.PT := T#130s;	// changed from := T#100s; (according to email 26.2.2020)
	END_IF;
	xTON_FA_T88();

	OUT_GT.bGT1_Check := xTON_FA_T88.Q;

	M_STPch		:=	OUT_GT.tGT1_SafeDevice.Do
					AND OUT_GT.bGT1_Check
					AND NOT OUT_GT.bGT1_CheckOK
					AND NOT IN_GT.tPCGT_SafeDevOK.Di
					AND Para.bPCGT_SafeDevice_Exist;

	M_STGAS1	:=	OUT_GT.tGT1_SafeDevice.Do
					AND OUT_GT.bGT1_Check
					AND NOT OUT_GT.bGT1_CheckOK
					AND ((NOT IN_GT.tGT1_SafeDevOK.Di AND NOT AKT_Gastrecke1_2) OR
						 (NOT IN_GT.tGT1_1_SafeDevOK.Di AND AKT_Gastrecke1_2));

	M_STGAS1_2	:=	OUT_GT.tGT1_SafeDevice.Do
					AND OUT_GT.bGT1_Check
					AND NOT OUT_GT.bGT1_CheckOK
					AND NOT IN_GT.tGT1_2_SafeDevOK.Di
					AND AKT_Gastrecke1_2;

	M_STGAS1_3	:=	OUT_GT.tGT1_SafeDevice.Do
					AND OUT_GT.bGT1_Check
					AND NOT OUT_GT.bGT1_CheckOK
					AND NOT IN_GT.tGT1_3_SafeDevOK.Di
					AND AKT_Gastrecke1_3;

	M_STGAS1_4	:=	OUT_GT.tGT1_SafeDevice.Do
					AND OUT_GT.bGT1_Check
					AND NOT OUT_GT.bGT1_CheckOK
					AND NOT IN_GT.tGT1_4_SafeDevOK.Di
					AND AKT_Gastrecke1_4;

	OUT_GT.bGT1_CheckOK   := OUT_GT.tGT1_SafeDevice.Do AND OUT_GT.bGT1_Check;

	IF Para.iNum_GT1_Lines < 2 THEN
		OUT_GT.bGT1_SafeDevOK := IN_GT.tGT1_SafeDevOK.Di OR IN_GT.bSafeOUT_GT1_SafeDevOK;	//Release from gastrain 1, no gasline 1-4 		(* SAFETY PLC *)
	ELSE
		OUT_GT.bGT1_SafeDevOK := bGT1_SafeDevOK 		 OR IN_GT.bSafeOUT_GT1_SafeDevOK;	//Release from gastrain 1, with gasline 1-4 	(* SAFETY PLC *)
	END_IF;

	(* if number of gastrains is < 2 *)
	IF (NOT OUT_GT.bGT_TypSwhActive AND NOT OUT_GT.bGT_TypSwhActiveHalt) THEN
		OUT_GT.bGT2_Check   := TRUE;
		OUT_GT.bGT2_CheckOK := TRUE;
		M_STGAS2 			:= FALSE;
	ELSE
		xTP_FA_T89.IN := NOT xTP_TP_vorStart.Q
					 AND NOT xTP_TP_vorStart2.Q
					 AND     T94
					 AND   ((OUT_GT.bGT2_Check AND NOT MM2VIS.bMsg1029) OR bOMSS_MAT);
		xTP_FA_T89.PT := T#1s;
		xTP_FA_T89();
	    T89 := xTP_FA_T89.Q;
		OUT_GT.tGT2_SafeDevice.Do := NOT T89 AND NOT IN_GT.bSafetyPLC_Active;			(* SAFETY PLC *)

		(* Testing time gas train 2 *)
		xTON_FA_T90.IN := OUT_GT.tGT2_SafeDevice.Do AND T94 AND ((OUT_GT.bGT2_Check AND NOT MM2VIS.bMsg1029) OR bOMSS_MAT);
		IF bTestEnabled THEN
			xTON_FA_T90.PT := T#1s;
		ELSE
			xTON_FA_T90.PT := T#130s;
		END_IF;
		xTON_FA_T90();
		OUT_GT.bGT2_Check := xTON_FA_T90.Q;

		M_STGAS2            := OUT_GT.tGT2_SafeDevice.Do AND OUT_GT.bGT2_Check AND NOT OUT_GT.bGT2_CheckOK AND NOT IN_GT.tGT2_SafeDevOK.Di;
		OUT_GT.bGT2_CheckOK := OUT_GT.tGT2_SafeDevice.Do AND OUT_GT.bGT2_Check;
	END_IF;

	OUT_GT.bGT2_SafeDevOK := IN_GT.tGT2_SafeDevOK.Di OR IN_GT.bSafeOUT_GT2_SafeDevOK;														(* SAFETY PLC *)

	(* Gas safety device Prechamber *)
	OUT_GT.tPCGT_SafeDevice.Do	:= OUT_GT.tGT1_SafeDevice.Do AND Para.bPCGT_SafeDevice_Exist;

	OUT_GT.bPCGT_SafeDevOK		:= IN_GT.tPCGT_SafeDevOK.Di OR NOT Para.bPCGT_SafeDevice_Exist;

END_PROGRAM
```

#### pb5.var - Local variables
```iecst
(********************************************************************
 * COPYRIGHT -- INNIO Company
 ********************************************************************
 * Program: pb5
 * File: pb5.var
 * Author: 105051626
 * Created: April 19, 2012
 ********************************************************************
 * Local variables of program pb5
 ********************************************************************)
VAR
	T87 : BOOL; (*Gas train 1 check*)
	T89 : BOOL; (*Gas train 2 check*)
	T94 : BOOL; (*Quiscent current loop OK*)
	xTON_FA_T94 : TON;
	xTON_FA_T88 : TON;
	xTON_FA_T90 : TON;
	xTP_FA_T89 : TP;
	xTP_TP_vorStart : TP;
	xTP_TP_vorStart2 : TP;
	xTP_FA_87 : TP;
	xSR_GT_SafetyDevice2ndStartBlock : SR;
	xTOF_SafetyCheck_Run : TOF := (0);
	bDelayForGascheck : BOOL := 0;
	xTON_GC_T100 : TON;
	xTOF_RESET : TOF;
	xTOF_Shutdown : TOF;
	RS_GK : RS;
	bDem_SafeDevice1 : BOOL := FALSE; (*internal*)
	bDem_SafeDevice2 : BOOL := FALSE; (*internal*)
	bDem_SafeDevice3 : BOOL := FALSE; (*internal*)
END_VAR
```

### Program Logical/Gastrain/gasline1_4 (IEC) - gas train 1 with 4 lines

#### gasline1_4.st - Cyclic code
```iecst
(*******************************************************************************
AGGR: 	gas train 1 with 4 lines

This code is confidential and proprietary to the INNIO Company.
It may not be used in any form, or reproduced in any manner, without the express
written permission of the INNIO Company.
Copyright, INNIO Company, 2019

Customized modifications: -
------------------------

History:
-------
V3.30.0	10.11.2011		glantschnig	new Implementation
V03.90.00.00	20.02.2013	Denk	V3.30 changes inserted in modular software
V04.01.00.00	15.07.2014	Denk	bugfix M_STGAS1

Instructions for use:
--------------------

Outstandings:
------------
-
*******************************************************************************)
PROGRAM _CYCLIC

	Para.iNum_GT1_Lines;							//Anzahl Gaslinien auswählen

	Para.iNum_GT1_Lines := LIMIT(1,Para.iNum_GT1_Lines,4);

	IF Para.iNum_GT1_Lines = 1 THEN					//Bei einer Gaslinien, 2-4 deaktivieren
		AKT_Gastrecke1_2 := FALSE;
		AKT_Gastrecke1_3 := FALSE;
		AKT_Gastrecke1_4 := FALSE;
	ELSIF Para.iNum_GT1_Lines = 2 THEN				//Bei zwei Gaslinien, 3-4 deaktivieren
		AKT_Gastrecke1_2 := TRUE;
		AKT_Gastrecke1_3 := FALSE;
		AKT_Gastrecke1_4 := FALSE;
	ELSIF Para.iNum_GT1_Lines = 3 THEN				//Bei drei Gaslinien, 4 deaktivieren
		AKT_Gastrecke1_2 := TRUE;
		AKT_Gastrecke1_3 := TRUE;
		AKT_Gastrecke1_4 := FALSE;
	ELSIF Para.iNum_GT1_Lines = 4 THEN				//Bei vier Gaslinien, 2-4 aktivieren
		AKT_Gastrecke1_2 := TRUE;
		AKT_Gastrecke1_3 := TRUE;
		AKT_Gastrecke1_4 := TRUE;
	END_IF

	IF Para.iNum_GT1_Lines < 2 THEN   				(* Para.iNum_GT1_Lines  < 2 is NOT active (default)	*)
		RETURN; 									(* Para.iNum_GT1_Lines  > 1     active      			*)
	END_IF;

	(* Common OUT for Gastrain 1 safety device OK *)
	bGT1_SafeDevOK :=	(IN_GT.tGT1_1_SafeDevOK.Di 								//Release from Gastrain 1 lines 1 - 4
					AND (IN_GT.tGT1_2_SafeDevOK.Di OR NOT AKT_Gastrecke1_2)
					AND (IN_GT.tGT1_3_SafeDevOK.Di OR NOT AKT_Gastrecke1_3)
					AND (IN_GT.tGT1_4_SafeDevOK.Di OR NOT AKT_Gastrecke1_4));

	OUT_GT.tGT1_1_SafeDevice.Do := OUT_GT.tGT1_SafeDevice.Do;							//Anforderung Gasdichtekontrollgerät Gasstrecke 1 - Linie 1
	OUT_GT.tGT1_2_SafeDevice.Do := OUT_GT.tGT1_SafeDevice.Do AND AKT_Gastrecke1_2;		//Anforderung Gasdichtekontrollgerät Gasstrecke 1 - Linie 2
	OUT_GT.tGT1_3_SafeDevice.Do := OUT_GT.tGT1_SafeDevice.Do AND AKT_Gastrecke1_3;		//Anforderung Gasdichtekontrollgerät Gasstrecke 1 - Linie 3
	OUT_GT.tGT1_4_SafeDevice.Do := OUT_GT.tGT1_SafeDevice.Do AND AKT_Gastrecke1_4;		//Anforderung Gasdichtekontrollgerät Gasstrecke 1 - Linie 4

END_PROGRAM
```

### Program Logical/Gastrain/gmv_ber (IEC) - gmv_ber

#### gmv_berCyclic.st - Cyclic code
```iecst
(* BERECHNUNG GASMISCHVERHÄLTNIS

.....................___
VER	Datum/Name	Änderung
V170	21.03.02/LH	erstellt
V172	17.09.02/LH	korrigiert für AS 2.2
V173	16.10.02/LH	Filter eingebaut (Robitschko)
V183	14.10.03/LH	angepasst für Gasumschaltung neu
V190	18.06.04/LH	Vermeidung von Rundungsfehlern
V3.99	21-09-2013	Ganguly/Denk, generated for modular software
*)

PROGRAM _CYCLIC

	(* Gas mixing relation *)
	IF GU_TJ THEN
		xLCRPT1_FA_GMISCH.x     := OUT_GT.rGT_RatioMix;
		xLCRPT1_FA_GMISCH.t		:= 0.2;
		xLCRPT1_FA_GMISCH();
		OUT_GT.rGasMixingRatio 	:= xLCRPT1_FA_GMISCH.y;
	END_IF;

END_PROGRAM
```

#### gmv_ber.var - Local variables
```iecst
VAR
	xLCRPT1_FA_GMISCH : LCRPT1;
END_VAR
```

#### gmv_berInit.st - Initialization code
```iecst
(********************************************************************
 * COPYRIGHT -- INNIO Company
 ********************************************************************
 * Program: gmv_ber
 * File: gmv_berInit.st
 * Author: 105051626
 * Created: May 10, 2012
 *******************************************************************)

PROGRAM _INIT
    xLCRPT1_FA_GMISCH.enable := TRUE;
	xLCRPT1_FA_GMISCH.t      := 0.2;
END_PROGRAM
```

### Program Logical/Gastrain/puffmini (IEC) - puffmini

#### puffminiCyclic.st - Cyclic code
```iecst
(* Verpuffungsminimierung, Freigabe Gasventile

VER	Date/Name	New
V0.10	29.06.07/Wa	generated
V0.20	20.02.08/LH	implemented into X20-system
V0.20.1	25.03.08/LH	renamed task from "puffmini_tc1" to "puffmini",
 			        name has to be maximum 8 characters!
V2.32.0	16.06.2008	lettenbichler	RUHE_M, RUHE_A removed, PILZ-SIGMA=standard
V2.33.0	17.07.2008	lettenbichler	GASV1_1, GASV1_2 added
V2.34.0	14.10.2008	lettenbichler	ZM_FG3_GASV: AB_NS, IN_GT.bRel_Island added
.					FG1_GASV: DI_GEN_PT added
V2.50.0	29.01.2009 	lettenb.		DI_GEN_PT -> IN_GT.tGenPrctTrip_TC2
.	    10.02.2009	puff_mini removed
V3.20.0	01.07.2010	lettenb.		port injection added
.			        maier (BuR)	DI_GCB_ON_TC1 replaced with GCB_ON_TC1
.			        maier (BuR)	DI_MCB_ON_TC1 replaced with IN_GT.tMCB_On_TC2
.	    21.10.2010  lettenb.    OUT_GT.tPCG_GV_DelOpen added
V3.99.0	21-09-2013	Ganguly/Denk	generated for modular software
V3.99.1 20.02.2013	Denk	V3.30 changes inserted
V3.99.2	20.02.2013	Denk 	Bugfix IN_GT.bMnsOK added in (IN_GT.tMnsOk_TC2.Di AND IN_GT.bMnsOk)

V04.03.00	13.11.2014	Denk		Bugfix, OUT_GT.tGV1_line1_Open.Do - OUT_GT.tGV1_line4_Open.Do added
			08.01.2015	Denk		Porting J920 to XT4
			31.03.2015	Denk 		Bugfix, assignment of OUT_GT.tGV1_line3_Open.Do, OUT_GT.tGV1_line4_Open.Do
V4.04.00	19.09.2016	Perktold	Bypass für FG-Gasventile bei Öffnen des GCB durch "tGrC_DCon.Do"
V4.05.00	08.01.2018	Denk		J-Maps finding, IN_GT.bEng_Start changed to IN_GT.bEng_Start_TC2
V4.12.00	10.03.2023	Perktold 	Bugfix - Bypass für FG-Gasventile bei Öffnen des GCB durch "tGrC_DCon.Do"
V4.13.00	30.11.2023	Goenczi 	Hold gas valve open in special cases, e.g. GCB at Customer
V4.14.00	22.11.2024	Schmidt 	Added pre chamber gas bypass valve logic (load acceptance improvements)
			09.04.2025	Perktold	Added GV3_Open and GV4_Open for SafetyPLC inputs
V4.25.00	14.01.2026	Tinello		Added DCGA output for SafetyPLC
*)

PROGRAM _CYCLIC

	xGR_MAXR_M_DR_ODR.In := IN_GT.rN_EngAct;
	xGR_MAXR_M_DR_ODR.Gw := Para.rN_EOP_Lim1;
	xGR_MAXR_M_DR_ODR.Hy := 10.0;
	xGR_MAXR_M_DR_ODR();
	M_DR_ODR := IN_GT.tPB2MM.bParaSetupOk AND xGR_MAXR_M_DR_ODR.Q;

	xGR_MAXR_FA_AN_FGPUFF.In := IN_GT.rP_Act_Norm_Filt;
	xGR_MAXR_FA_AN_FGPUFF.Hy := Para.rP_DeflagPrct_Hy;
	xGR_MAXR_FA_AN_FGPUFF.Gw := Para.rDeflagPrct_Lim;
	xGR_MAXR_FA_AN_FGPUFF();
	AN_FGPUFF := xGR_MAXR_FA_AN_FGPUFF.Q AND IN_GT.tPB2MM.bParaSetupOk;

	(* speed limit *)
	xGR_MAXR_D1400(In:= IN_GT.rN_EngAct, Gw:= (Para.rN_EngNom - 100.0), Hy:= 10.0);
	M_D1400	:= xGR_MAXR_D1400.Q AND IN_GT.tPB2MM.bParaSetupOk;

	(* differential protection monitoring release *)
	xSR_FG_DIFFUW(SET1  := M_D1400,
				  RESET := IN_GT.bEng_Start_TC2 OR (NOT M_D1400 AND NOT OUT_GT.bGV_On AND NOT IN_GT.bEng_Dem AND NOT IN_GT.tGCB_On.Di));

	(* release gas valves by gcb monitoring:
	differential protection, earth failure, overload/short circuit/Kurzschluss, gen.protection trip(onsite) *)
	FG1_GASV :=(IN_GT.tDiffPrct_TC2.Di OR (NOT xSR_FG_DIFFUW.Q1 AND Para.bPF_CosPCtr_Diff_Ena))
			AND IN_GT.tGndFailure_TC2.Di
			AND IN_GT.tOlShortCirc_TC2.Di
			AND IN_GT.tGenPrctTrip_TC2.Di;

	(* Release gas valve with Main OK (depending on installation) *)
	FG2_GASV := ((IN_GT.tMnsOk_TC2.Di AND IN_GT.bMnsOk) OR IN_GT.bRel_Island OR IN_GT.bRel_IslandAfMITime OR NOT Para.bSyActive OR Para.bMIF_Enable)
				AND IN_GT.bRelEngOpFromSy;

	(* Detect external switch GS or external switch off mains circuit breaker ( depending on installation) *)
	xF_TRIG_FA_GSAUS.CLK := IN_GT.tGCB_On_TC2.Di;
	xF_TRIG_FA_GSAUS();

	xF_TRIG_FA_NSAUS.CLK := IN_GT.tMCB_On_TC2.Di;
	xF_TRIG_FA_NSAUS();

	xTP_GrC(IN := NOT IN_GT.tGrC_DCon.Do, PT := tGrC_Bypass);

	(*GCB opening by Customer without GCB command off from DiaNe - GCB control at Customer*)
	IF IN_GT.bGCB_by_Customer AND xF_TRIG_FA_GSAUS.Q THEN
		IF (NOT IN_GT.tP_Lo.Do AND (IN_GT.rP_Act_Norm_Filt < 0.15))		//Power below GCB opening limit
			OR ((xEngType.Type < 6) AND Para.bMisfCont)					//Type 2/3/4 engine with activated Misfire Control
			OR ((xEngType.Type = 6) AND Para.bP_LoadReject_Active)		//Type 6 engine with activated LoadRejection package incl. blow off valve
		THEN
			bHOLD_FG3_GASV	:= 	TRUE;
		ELSE
			bHOLD_FG3_GASV	:= 	FALSE;
		END_IF;
	ELSE
		bHOLD_FG3_GASV	:= 	FALSE;
	END_IF;
	ZM_FG3_GASV := (((xF_TRIG_FA_GSAUS.Q AND NOT xTP_GrC.Q) AND IN_GT.tGCB_COf.Do) AND NOT bHOLD_FG3_GASV) OR
	               (xF_TRIG_FA_NSAUS.Q AND IN_GT.tMCB_COf.Do AND NOT IN_GT.bRel_Island);

	FG3_GASV := NOT ZM_FG3_GASV;

	(* Release gas valve (--> Blocking module ) *)
	xTON_FA_FG_GASV.IN := FG1_GASV AND FG2_GASV AND FG3_GASV;
	xTON_FA_FG_GASV.PT := T#1s;
	xTON_FA_FG_GASV();
	OUT_GT.tGV_Rel.Do  := xTON_FA_FG_GASV.Q;

	(* Release port injection *)
	OUT_GT.bPortInject_Rel := (GASV1_TC3 OR GASV2_TC3) AND OUT_GT.tGV_Rel.Do;

	(* Close gas valves with Speed < parameter and release gas valves for port injection *)		//Porting J920 to XT4, with XT3: 20.11.2014 Tinello GR_MAX_GASV removed
//	xGR_MAXR_GASV.In := IN_GT.rN_EngAct;
//	xGR_MAXR_GASV.Gw := Para.rN_GV_CloseLimMin;
//	xGR_MAXR_GASV.Hy := 10;
//	xGR_MAXR_GASV();
	FG_GASV_PI       := OUT_GT.bPortInject_Rel;													//Porting J920 to XT4, with XT3: 20.11.2014 Tinello GR_MAX_GASV removed

	(* Arrange open outputs *)
	(* Gas valve 1 *)
	OUT_GT.tGV1_Open.Do 	:= GASV1_TC3 AND ((OUT_GT.tGV_Rel.Do AND NOT xEngType.Type9) OR (FG_GASV_PI AND xEngType.Type9 ));
	OUT_GT.tGV1_1_Open.Do 	:= GASV1_TC3 AND ((OUT_GT.tGV_Rel.Do AND NOT xEngType.Type9) OR (FG_GASV_PI AND xEngType.Type9)) AND IN_GT.bSCO_Rel_GV1;
	OUT_GT.tGV1_2_Open.Do 	:= GASV1_TC3 AND ((OUT_GT.tGV_Rel.Do AND NOT xEngType.Type9) OR (FG_GASV_PI AND xEngType.Type9)) AND IN_GT.bSCO_Rel_GV2 AND M_DR_ODR;
	(* Gas valve 1 - lines 1-4 *)
	OUT_GT.tGV1_line1_Open.Do 	:= OUT_GT.tGV1_Open.Do;
	OUT_GT.tGV1_line2_Open.Do 	:= OUT_GT.tGV1_Open.Do AND AKT_Gastrecke1_2;
	OUT_GT.tGV1_line3_Open.Do 	:= OUT_GT.tGV1_Open.Do AND AKT_Gastrecke1_3;
	OUT_GT.tGV1_line4_Open.Do 	:= OUT_GT.tGV1_Open.Do AND AKT_Gastrecke1_4;
	(* Gas valve 2 *)
	OUT_GT.tGV2_Open.Do 	:= GASV2_TC3 AND ((OUT_GT.tGV_Rel.Do AND NOT xEngType.Type9) OR (FG_GASV_PI AND xEngType.Type9));

	(* Gas velve 3/4 - prepared for SafetyPLC input but not used*)
	OUT_GT.tGV3_Open.Do 	:= FALSE;
	OUT_GT.tGV4_Open.Do 	:= FALSE;
	OUT_GT.tDCGA_GV_Open.Do := FALSE;									(* SAFETY PLC *)

	(* Pre chamber gas valve  *)
	OUT_GT.tPCG_GV_Open.Do := VKGV_TC3 AND OUT_GT.tGV_Rel.Do;

	(* Pre chamber gas valve stepped power on (in-rush current) *)
	xTON_VKGK2.IN := VKGV_TC3 AND OUT_GT.tGV_Rel.Do;
	xTON_VKGK2.PT := T#0.5s;
	xTON_VKGK2();
	OUT_GT.tPCG_GV_DelOpen.Do := xTON_VKGK2.Q;

	(* Pre chamber gas bypass valve - START *)
	(* First-order low-pass filter of measured power *)
	xLCRPT1_P_Act_Filt.enable		:= TRUE;
	xLCRPT1_P_Act_Filt.x			:= IN_GT.tP_Act[1].Unfilt;
	xLCRPT1_P_Act_Filt.t			:= MAX(0.0001, rTau_P_Act_Filt);
	xLCRPT1_P_Act_Filt.y_set 		:= IN_GT.tP_Act[1].Unfilt;
	xLCRPT1_P_Act_Filt.set 			:= NOT IN_GT.tGCB_On_TC2.Di;
	xLCRPT1_P_Act_Filt();

	(* Check if the charge pressure is below the barometric pressure *)
	xGR_MINR_p2s_pbaro(In := IN_GT.rPr_Ch_P2s_Avg_UF, Gw := IN_GT.rPr_Baro_Internal, Hy := rHyst_GR_MINR_p2s_pbaro);
	(* Compare filtered and unfiltered power to detect a load acceptance *)
	xR_TRIG_P_Compare(CLK := ((IN_GT.tP_Act[1].Unfilt / MAX(0.0001, IN_GT.rP_Nom)) - (xLCRPT1_P_Act_Filt.y / MAX(0.0001, IN_GT.rP_Nom))) > rP_Norm_Act_Filt_Thresh);
	xTP_P_Compare(IN := xR_TRIG_P_Compare.Q, PT := tP_Compare);

	(* If the charge pressure is below the barometric pressure and a load acceptance is detected, the pre chamber gas bypass valve shall be opened.
	   The pre chamber gas bypass valve shall be closed after the load acceptance, once the volume change in the V-room is reduced again or if the boost pressure exceeds the barometric pressure *)
	IF Para.bPCG_BPV_Active AND xEngType.Type6 AND xOpMode.Island AND IN_GT.tGCB_On_TC2.Di AND OUT_GT.tPCG_GV_Open.Do AND xGR_MINR_p2s_pbaro.Q THEN
		IF xTP_P_Compare.Q THEN
			OUT_GT.tPCG_BPV_Open.Do := TRUE;
		ELSIF OUT_GT.tPCG_BPV_Open.Do AND (IN_GT.rFlow_VR_TJ < rFlow_VR_Thresh) THEN
			OUT_GT.tPCG_BPV_Open.Do := FALSE;
		END_IF;
	ELSE
		OUT_GT.tPCG_BPV_Open.Do := FALSE;
	END_IF;
	(* Pre chamber gas bypass valve - END *)

END_PROGRAM
```

#### puffmini.var - Local variables
```iecst
VAR
	ZM_FG3_GASV : BOOL := 0;
	FG_GASV_PI : BOOL;
	FG3_GASV : BOOL := 0;
	FG1_GASV : BOOL;
	FG2_GASV : BOOL := 0;
	xF_TRIG_FA_NSAUS : F_TRIG;
	xF_TRIG_FA_GSAUS : F_TRIG;
	xGR_MAXR_FA_AN_FGPUFF : GR_MAXR;
	xTON_FA_FG_GASV : TON;
	xTON_VKGK2 : TON;
	xGR_MAXR_M_DR_ODR : GR_MAXR;
	xGR_MAXR_D1400 : GR_MAXR;
	M_D1400 : BOOL;
	xSR_FG_DIFFUW : SR;
	xTP_GrC : TP;
	tGrC_Bypass : TIME := T#250ms;
	bHOLD_FG3_GASV : BOOL; (*hold FG3_GASV at GCB opening in special cases - new 14/10/2020*)
	xLCRPT1_P_Act_Filt : LCRPT1; (* FuB first-order low-pass filter for power *)
	rTau_P_Act_Filt : REAL := 2.0; (* Filter time constant [s] *)
	xGR_MINR_p2s_pbaro : GR_MINR; (* FuB for comparison of charge and ambient pressure *)
	rHyst_GR_MINR_p2s_pbaro : REAL := 0.05; (* Hysteresis for comparison of charge and ambient pressure [bar] *)
	rP_Norm_Act_Filt_Thresh : REAL := 0.08; (* Threshold comparison of unfilt. and filt. power to detect load step [PercentPnom] *)
	xR_TRIG_P_Compare : R_TRIG; (* FuB power comparison *)
	xTP_P_Compare : TP; (* Pulse for load step detection *)
	tP_Compare : TIME := T#500ms; (* Minimum duration of PCG BPV opening after load step detection [ms] *)
	rFlow_VR_Thresh : REAL := 0.15; (* Threshold for PCG BPV closing based on volume change V-room [m3/s] *)
END_VAR
```

### Program Logical/Gastrain/vkgverd (IEC) - vkgverd

#### vkgverdCyclic.st - Cyclic code
```iecst
(* Vorkammergasverdichter

.....................___
VER	Datum/Name	Änderung
V0.1	26.01.99/Pa	erstellt
V160	04.12.01/LH	Ansteuerung Entlastungsventil verzögert
V161	11.03.02/LH	vkgverd	Ausgang Entlastungsventil umgedreht
V170	12.03.02/LH	Vorkammergasdruckstörungen aufbereitet
V172	11.07.02/LH	überarbeitet
V173	13.11.02/LH	Einlesen des Analogeinganges in pb17 verlegt
V2071	02.02.05/LH	Bezeichnungen überarbeitet
V2071b	28.06.05/LH	Netzwerkkommentare korrigiert
V2071c	20.09.05/LH	Variable "Para.bPr_PCG_GC_Active" eingeführt (für Überwachung in pb10)
V2072	16.11.05/LH	Grenzwert Verdichter EIN: 2,80 bar --> 3,00 bar
 			        Grenzwert Verdichter AUS: 3,80 bar --> 3,70 bar
V190	30.08.04/LH	Grenzwerte einstellbar und auf Standardstörungen
V210	05.01.06/LH	angepasst für V210
V2201	17.07.07/LH	Erweiterungen für wassergekühlten Verdichter
 			        Abstellung bei Ölstand minimum
  	    23.07.07/LH	Verlängerung Nachkühlzeit Verdichter auf 30s (lt. Hersteller)
V03.99.00.00	21.09.2013	Ganguly	generated for modular software
V04.00.01.00 	17.05.14	Denk	NOT MM2VIS.bMsg3315;
V04.01.01.00 	07.10.14	Denk	Adicom Pre-chamber gas compressor logic added
*)

PROGRAM _CYCLIC

	IF Para.bPr_PCG_GC_Active THEN

		(* Set point pressure pre-chamber gas compressor minimum *)
		xGR_MINR_FA_AN_VKMIN.In := IN_GT.tPr_PCG.Ai;
		xGR_MINR_FA_AN_VKMIN.Gw := Para.rPr_PCG_GC_LimMin;
		xGR_MINR_FA_AN_VKMIN.Hy := Para.rPr_PCG_GC_HyMin;
		xGR_MINR_FA_AN_VKMIN();
		AN_VKMIN := xGR_MINR_FA_AN_VKMIN.Q AND IN_GT.tPB2MM.bParaSetupOk;

		(* Set point pre-chamber gas compressor ON *)
		xGR_MINR_FA_AN_VKEIN.In := IN_GT.tPr_PCG.Ai;
		xGR_MINR_FA_AN_VKEIN.Gw := Para.rPr_PCG_GC_LimOff;
		xGR_MINR_FA_AN_VKEIN.Hy := 0.1;						//#4 old code: 1000 --> 10.00 bar, #6 FA_AN_VKEIN.Hy old code 10 --> 0.1 bar
		xGR_MINR_FA_AN_VKEIN();
		AN_VKEIN := xGR_MINR_FA_AN_VKEIN.Q AND IN_GT.tPB2MM.bParaSetupOk;

		(* Set point pre chamber gas compressor - OFF *)
		xGR_MAXR_FA_AN_VKAUS.In := IN_GT.tPr_PCG.Ai;
		xGR_MAXR_FA_AN_VKAUS.Gw := Para.rPr_PCG_GC_LimOn;
		xGR_MAXR_FA_AN_VKAUS.Hy := 0.1;
		xGR_MAXR_FA_AN_VKAUS();
		AN_VKAUS := xGR_MAXR_FA_AN_VKAUS.Q AND IN_GT.tPB2MM.bParaSetupOk;

		(* Set point Pressure pre chamber gas compressor maximum *)
		xGR_MAXR_FA_AN_VKMAX.In := IN_GT.tPr_PCG.Ai;
		xGR_MAXR_FA_AN_VKMAX.Gw := Para.rPr_PCG_GC_LimMax;
		xGR_MAXR_FA_AN_VKMAX.Hy := Para.rPr_PCG_GC_HyMax;
		xGR_MAXR_FA_AN_VKMAX();
		AN_VKMAX := xGR_MAXR_FA_AN_VKMAX.Q AND IN_GT.tPB2MM.bParaSetupOk;

	ELSE
		AN_VKMIN := FALSE;
		AN_VKMAX := FALSE;
		AN_VKEIN := FALSE;
		AN_VKAUS := FALSE;
	END_IF;

	(* Release monitoring pressure prechamber gas compressor *)
	xTON_FA_UW_VKGD.IN := OUT_GT.tPr_PCG_GC_Dem.Do ;
	xTON_FA_UW_VKGD.PT := T#1m;
	xTON_FA_UW_VKGD();
	UW_VKGD := xTON_FA_UW_VKGD.Q;

	(* Pressure Pre-chamber gas compressor minimum *)
	VKGD_MIN :=  (UW_VKGD OR IN_GT.tEng_Run.Do) AND AN_VKMIN AND IN_GT.tPr_PCG.GoodQual;

	(* Pressure Pre-chamber gas compressor maximum *)
	VKGD_MAX := AN_VKMAX;

	(* Stop gas compressor because of: *)
	(* - Emergency-OFF, Gas alarm, Gas pre-alarm, Fire alarm, .... *)
	STOER := NOT IN_GT.bMsg1054 AND NOT IN_GT.bMsg1052 AND NOT IN_GT.bMsg1053 AND NOT IN_GT.bMsg1031;
	(* - Pre-chamber gas pressure minimum, pressure pre chamber gas compressor maximum, measure signal failure
	pre-chamber gas compressor pressure *)
	STOER := STOER AND NOT MM2VIS.bMsg1095 AND NOT MM2VIS.bMsg3309 AND NOT MM2VIS.bMsg3308;
	(* - Oil level minimum pre chamber gas compressor *)
	STOER := STOER AND NOT MM2VIS.bMsg3315;

	(* Pre-chamber gas compressor *)
	IF Para.bPr_PCG_GC_Active THEN			(* demand pre chamber gas compressor - control and monitoring by GEJ *)
		OUT_GT.tPr_PCG_GC_Dem.Do := STOER
								    AND (AN_VKEIN OR (NOT AN_VKAUS AND OUT_GT.tPr_PCG_GC_Dem.Do))
									AND (IN_GT.bEng_Dem OR M_DREHZ);
	ELSE									(* demand pre chamber gas compressor -  compressor package*)
		OUT_GT.tPr_PCG_GC_Dem.Do := STOER
									AND (IN_GT.bEng_Dem OR M_DREHZ);
	END_IF;

	(* Switch-ON unloading valve *)
	xTOF_FA_ENTLV.IN := NOT OUT_GT.tPr_PCG_GC_Dem.Do ;
	xTOF_FA_ENTLV.PT := T#0.5s;
	xTOF_FA_ENTLV();
	ENTLV := xTOF_FA_ENTLV.Q;

	xTON_FA_ENTL_V.IN := ENTLV;
	xTON_FA_ENTL_V.PT := T#0.5s;
	xTON_FA_ENTL_V();
	OUT_GT.tPCG_DemReliefValve.Do := NOT xTON_FA_ENTL_V.Q;

	(* Auxilliary compressor *)
	xTOF_FA_HBT_VERD.IN := OUT_GT.tPr_PCG_GC_Dem.Do ;
	xTOF_FA_HBT_VERD.PT := T#30s;
	xTOF_FA_HBT_VERD();

	OUT_GT.tPCG_DemValCW.Do   := xTOF_FA_HBT_VERD.Q;
	OUT_GT.tPCG_DemCoolFan.Do := xTOF_FA_HBT_VERD.Q;

END_PROGRAM
```

#### vkgverd.var - Local variables
```iecst
VAR
	STOER : BOOL := 0; (* Störung Vorkammergasverdichter *)
	ENTLV : BOOL;
	UW_VKGD : BOOL;
	AN_VKMIN : BOOL;
	AN_VKMAX : BOOL;
	AN_VKEIN : BOOL;
	AN_VKAUS : BOOL;

	xGR_MAXR_FA_AN_VKAUS : GR_MAXR;
	xGR_MAXR_FA_AN_VKMAX : GR_MAXR;
	xGR_MINR_FA_AN_VKMIN : GR_MINR;
	xGR_MINR_FA_AN_VKEIN : GR_MINR;

	xTOF_FA_HBT_VERD : TOF;
	xTOF_FA_ENTLV : TOF;
	xTON_FA_UW_VKGD : TON;
	xTON_FA_ENTL_V : TON;

END_VAR
```

### Program Logical/Gastrain/CommonGT (IEC) - Common alarms and signal generation for GT module

#### CommonGTCyclic.st - Cyclic code
```iecst
(*******************************************************************************
CommonGT	 			 common functions

This code is confidential and proprietary to the INNIO Company.
It may not be used in any form, or reproduced in any manner,
without written permission of the INNIO Company.
Copyright, INNIO Company, 2019

Customized modifications: -
------------------------

History:
-------
V3.99		21-09-2013	Ganguly/Denk, 	generated for modular software
			23.04.2013	lettenb.		logic for 1085, 3315 moved to MsgGT
V04.00.01	11.03.2014	Denk			gas type 123 Display changed 1=1, 3=3,..!
V04.03.00 	03.02.2015  Denk			Porting J920 FOR XT4
V04.04.00	21.07.2016	Denk			Bugfix, Display on Visu
V04.11.00	21.10.2021	Zuschnig		Update prechamber gas train power reduction
V04.13.00	05.12.2023	Zuschnig		Update prechamber gas train power reduction in island mode
V04.14.00	11.12.2024	Zuschnig		Prechamber gas train power reduction in island mode - W9387 only if reduced power < 1

Instructions for use:
--------------------

Outstandings:
------------

(*******************************************************************************)

PROGRAM _CYCLIC

	(* Motortype *)
	xEngType.Motortype := INT_TO_UINT(Para.iEng_Motortype);
	xEngType();

	(* Engine operating mode *)
	xOpMode(in := IN_GT.iSt_OpMode);

	(* Operation mode selector switch in manual, auto or probe mode*)
	bOMSS_MAT := (IN_GT.iIdx_OMSS = 1) OR (IN_GT.iIdx_OMSS = 2) OR (IN_GT.iIdx_OMSS = 3);

	(* M_DREHZ signal generation *)
	xGR_MAXR_FA_AN_DREHZ.In := IN_GT.rN_EngAct;
	xGR_MAXR_FA_AN_DREHZ.Hy := Para.rN_EngStart_HyHi;
	xGR_MAXR_FA_AN_DREHZ.Gw := Para.rN_EngStart_LimHi;
	xGR_MAXR_FA_AN_DREHZ();
	xTOF_FA_M_DREHZ.IN := xGR_MAXR_FA_AN_DREHZ.Q AND IN_GT.tPB2MM.bParaSetupOk;
	xTOF_FA_M_DREHZ.PT := T#10s;
	xTOF_FA_M_DREHZ();
	M_DREHZ := xTOF_FA_M_DREHZ.Q;

	(* Release gas pressure monitoring - include relese gas monitoring form external set customized logic for FG_GDRUW_ext *)
	FG_GDRUW := IN_GT.tEng_Run.Do
			OR (IN_GT.bEng_Aux_Dem AND NOT IN_GT.bEng_Start AND NOT OUT_GT.bGV_On AND bP_GT_RelMonExt);

	(* Selection of gassort in dependence of the gassort bit´s *)
	TON_SecondTick(IN:=NOT TON_SecondTick.Q, PT:= T#800ms);							(* timer for 1 second tick  = 800ms + 2 task class cycles *)

	IF		(IN_GT.bGasTypMix1_2_Act AND NOT IN_GT.bGasTyp3_Act)	THEN	OUT_GT.iIdx_Gtyp_Dem := 0;			(* gassort 0 *)
	ELSIF	IN_GT.bGasTyp2_Act = TRUE 								THEN	OUT_GT.iIdx_Gtyp_Dem := 2;			(* gassort 2 *)
	ELSIF 	IN_GT.bGasTyp3_Act = TRUE								THEN	OUT_GT.iIdx_Gtyp_Dem := 3;			(* gassort 3 *)
	ELSIF 	IN_GT.bGasTyp4_Act = TRUE								THEN	OUT_GT.iIdx_Gtyp_Dem := 4;			(* gassort 4 *)
	ELSE 	OUT_GT.iIdx_Gtyp_Dem := 1;																			(* otherwise gassort 1 *)
	END_IF;
	IF bCrossOver THEN
		OUT_GT.iIdx_Gtyp_Dem := 0;				(* gassort 0 *)
	END_IF;

	(* Gastype selection for VISU display *)
	(* create extended gas type selection *)
	CASE OUT_GT.iIdx_Gtyp_Dem OF
	1:	MM2VIS.iIdx_Gtyp_Act := 1;				(* gas type 1 *)
	2:	MM2VIS.iIdx_Gtyp_Act := 2;				(* gas type 2 *)
	3:	MM2VIS.iIdx_Gtyp_Act := 3;				(* gas type 3 *)
	4:	MM2VIS.iIdx_Gtyp_Act := 4;				(* gas type 4 *)
	ELSE
		IF OUT_GT.bGasMixingActive THEN
			IF OUT_GT.bGT_Ipol12Active THEN
				MM2VIS.iIdx_Gtyp_Act := 123;	(* gas type 1_2/3 *)
			ELSE
				MM2VIS.iIdx_Gtyp_Act := 13;		(* gas type 1/3 *)
			END_IF;
		ELSE
			IF IN_GT.bGasTyp3_Act = TRUE THEN
				MM2VIS.iIdx_Gtyp_Act := 3;		(* gas type 3 *)
			ELSE
				MM2VIS.iIdx_Gtyp_Act := 12;		(* gas type 1_2 *)
			END_IF;
		END_IF;
	END_CASE;

	(* power reduction according low pressure in pre chamber gas train *)
	OUT_GT.rPr_P2s_demand_PCGT	:=	IN_GT.tPr_PCGT.Ai + IN_GT.rPr_Baro_Internal - Para.rDPr_PCGT_Set - rPr_PCGT_PipeLoss;

	IF Para.bP_Red_Pr_PCG AND Para.bPr_PCGT_Active AND IN_GT.tPr_PCGT.GoodQual AND OUT_GT.tPCG_GV_Open.Do THEN
		OUT_GT.rP_Red_Pr_PCGT_Norm := LIMIT(0, (IN_GT.rP_el_max_red_PCGT / MAX(1, IN_GT.rP_Nom)), 1.0);
	ELSE
		OUT_GT.rP_Red_Pr_PCGT_Norm := 1.0;
	END_IF;

	IF xOpMode.NetP AND Para.bPr_PCGT_Active AND (OUT_GT.rP_Red_Pr_PCGT_Norm < IN_GT.rP_Set_Min_Norm) THEN
		bPowerMin_PCGT	:= TRUE;
	ELSIF xOpMode.Island AND Para.bPr_PCGT_Active AND (IN_GT.rPr_Ch_P2s_Avg > (IN_GT.tPr_PCGT.Ai + IN_GT.rPr_Baro_Internal - Para.rDPr_PCGT_Set)) AND NOT Para.bSA_PI_Active THEN
		bPowerMin_PCGT	:= TRUE;
	ELSE
		bPowerMin_PCGT	:= FALSE;
	END_IF;

	IF xOpMode.Island AND Para.bPr_PCGT_Active AND (OUT_GT.rP_Red_Pr_PCGT_Norm < IN_GT.rP_Act_Norm_Filt) AND NOT Para.bSA_PI_Active AND (OUT_GT.rP_Red_Pr_PCGT_Norm < 1.0) THEN
		bMsg9387_Set := TRUE;
	ELSE
		bMsg9387_Set := FALSE;
	END_IF;

	(* release main gas valve *)
	FG_HGV := NOT IN_GT.bMsg1053 AND NOT IN_GT.bMsg1052 AND NOT IN_GT.bMsg1054 AND NOT IN_GT.bMsg1031
			AND IN_GT.tRelMainGVext.Di;

	(* Check if velocity is zero *)
	IF IN_GT.rN_EngAct > -0.01 AND IN_GT.rN_EngAct < 0.01 THEN
		bN_EngAct_IsZero := TRUE;
	ELSE
		bN_EngAct_IsZero := FALSE;
	END_IF;

END_PROGRAM
```

#### CommonGT.var - Local variables
```iecst
VAR
	xGR_MAXR_FA_AN_DREHZ : GR_MAXR;
	xTOF_FA_M_DREHZ : TOF;
	TON_SecondTick : TON; (* FUB 1 second timer tick *)
	rPr_PCGT_PipeLoss : REAL := 0.1; (* Pressure loss offset PCGT [bar] *)
END_VAR
```

### Program Logical/Gastrain/pb7 (IEC) - pb7
